  Call Extruder(591.82006)
  MoveL 2707 to (233.6, 37.71, 50.44) mm, rotated rx -180 ry 0 rz 180 deg; joints [-18.033, 13.455, 54.768, 41.267, 27.992, -37.77]
  MoveL 2708 to (233.6, 37.71, 50.44) mm, rotated rx -180 ry 0 rz 180 deg; joints [-18.033, 13.455, 54.768, 41.267, 27.992, -37.77]
  Call Extruder(592.02779)
  MoveL 2709 to (233.9, 37.89, 50.44) mm, rotated rx -180 ry 0 rz 180 deg; joints [-18.041, 13.521, 54.685, 41.26, 28.009, -37.759]
  MoveL 2710 to (233.9, 37.89, 50.44) mm, rotated rx -180 ry 0 rz 180 deg; joints [-18.041, 13.521, 54.685, 41.26, 28.009, -37.759]
  Call Extruder(592.23629)
  MoveL 2711 to (234.21, 38.07, 50.44) mm, rotated rx 180 ry 0 rz 180 deg; joints [-18.049, 13.588, 54.602, 41.254, 28.027, -37.748]
  MoveL 2712 to (234.21, 38.07, 50.44) mm, rotated rx 180 ry 0 rz 180 deg; joints [-18.049, 13.588, 54.602, 41.254, 28.027, -37.748]
  Call Extruder(592.41583)
  MoveL 2713 to (234.45, 38.24, 50.44) mm, rotated rx 180 ry 0 rz 180 deg; joints [-18.06, 13.643, 54.532, 41.254, 28.043, -37.744]
  MoveL 2714 to (234.45, 38.24, 50.44) mm, rotated rx 180 ry 0 rz 180 deg; joints [-18.06, 13.643, 54.532, 41.254, 28.043, -37.744]
  Call Extruder(592.74925)
  MoveL 2715 to (234.9, 38.57, 50.44) mm, rotated rx -180 ry 0 rz -180 deg; joints [-18.079, 13.746, 54.404, 41.255, 28.075, -37.737]
  MoveL 2716 to (234.9, 38.57, 50.44) mm, rotated rx -180 ry 0 rz -180 deg; joints [-18.079, 13.746, 54.404, 41.255, 28.075, -37.737]
  Call Extruder(593.08385)
  MoveL 2717 to (235.35, 38.9, 50.44) mm, rotated rx 180 ry 0 rz -180 deg; joints [-18.099, 13.849, 54.274, 41.255, 28.107, -37.729]
  Call Extruder(593.91180)
  MoveL 2718 to (236.39, 39.81, 50.44) mm, rotated rx -180 ry 0 rz 180 deg; joints [-18.16, 14.097, 53.963, 41.28, 28.192, -37.731]
  Call Extruder(594.73974)
  MoveL 2719 to (237.3, 40.85, 50.44) mm, rotated rx -180 ry 0 rz 180 deg; joints [-18.24, 14.33, 53.668, 41.337, 28.287, -37.762]
  Call Extruder(594.90704)
  MoveL 2720 to (237.47, 41.07, 50.44) mm, rotated rx -180 ry 0 rz 180 deg; joints [-18.258, 14.375, 53.612, 41.353, 28.307, -37.773]
  MoveL 2721 to (237.47, 41.07, 50.44) mm, rotated rx -180 ry 0 rz 180 deg; joints [-18.258, 14.375, 53.612, 41.353, 28.307, -37.773]
  Call Extruder(595.24045)
  MoveL 2722 to (237.79, 41.52, 50.44) mm, rotated rx 180 ry 0 rz 180 deg; joints [-18.295, 14.464, 53.499, 41.385, 28.347, -37.794]
  MoveL 2723 to (237.79, 41.52, 50.44) mm, rotated rx 180 ry 0 rz 180 deg; joints [-18.295, 14.464, 53.499, 41.385, 28.347, -37.794]
  Call Extruder(595.57268)
  MoveL 2724 to (238.12, 41.98, 50.44) mm, rotated rx 180 ry 0 rz 180 deg; joints [-18.332, 14.554, 53.385, 41.417, 28.388, -37.814]
  MoveL 2725 to (238.12, 41.98, 50.44) mm, rotated rx 180 ry 0 rz 180 deg; joints [-18.332, 14.554, 53.385, 41.417, 28.388, -37.814]
  Call Extruder(595.69039)
  MoveL 2726 to (238.22, 42.15, 50.44) mm, rotated rx 180 ry 0 rz 180 deg; joints [-18.346, 14.583, 53.348, 41.432, 28.403, -37.825]
  MoveL 2727 to (238.22, 42.15, 50.44) mm, rotated rx 180 ry 0 rz 180 deg; joints [-18.346, 14.583, 53.348, 41.432, 28.403, -37.825]
  Call Extruder(595.89811)
  MoveL 2728 to (238.4, 42.45, 50.44) mm, rotated rx -180 ry 0 rz 180 deg; joints [-18.373, 14.635, 53.282, 41.458, 28.429, -37.843]
  MoveL 2729 to (238.4, 42.45, 50.44) mm, rotated rx -180 ry 0 rz 180 deg; joints [-18.373, 14.635, 53.282, 41.458, 28.429, -37.843]
  Call Extruder(596.10507)
  MoveL 2730 to (238.57, 42.75, 50.44) mm, rotated rx -180 ry 0 rz -180 deg; joints [-18.399, 14.687, 53.216, 41.485, 28.456, -37.862]
  MoveL 2731 to (238.57, 42.75, 50.44) mm, rotated rx -180 ry 0 rz -180 deg; joints [-18.399, 14.687, 53.216, 41.485, 28.456, -37.862]
  Call Extruder(596.31124)
  MoveL 2732 to (238.75, 43.06, 50.44) mm, rotated rx 180 ry 0 rz 180 deg; joints [-18.425, 14.739, 53.15, 41.511, 28.483, -37.881]
  MoveL 2733 to (238.75, 43.06, 50.44) mm, rotated rx 180 ry 0 rz 180 deg; joints [-18.425, 14.739, 53.15, 41.511, 28.483, -37.881]
  Call Extruder(596.49292)
  MoveL 2734 to (238.89, 43.34, 50.44) mm, rotated rx 180 ry 0 rz 180 deg; joints [-18.45, 14.783, 53.094, 41.537, 28.507, -37.9]
  MoveL 2735 to (238.89, 43.34, 50.44) mm, rotated rx 180 ry 0 rz 180 deg; joints [-18.45, 14.783, 53.094, 41.537, 28.507, -37.9]
  Call Extruder(596.65093)
  MoveL 2736 to (239, 43.58, 50.44) mm, rotated rx -180 ry 0 rz 180 deg; joints [-18.472, 14.819, 53.048, 41.563, 28.528, -37.919]
  MoveL 2737 to (239, 43.58, 50.44) mm, rotated rx -180 ry 0 rz 180 deg; joints [-18.472, 14.819, 53.048, 41.563, 28.528, -37.919]
  Call Extruder(596.80833)
  MoveL 2738 to (239.11, 43.83, 50.44) mm, rotated rx 180 ry 0 rz -180 deg; joints [-18.495, 14.854, 53.003, 41.588, 28.549, -37.939]
  MoveL 2739 to (239.11, 43.83, 50.44) mm, rotated rx 180 ry 0 rz -180 deg; joints [-18.495, 14.854, 53.003, 41.588, 28.549, -37.939]
  Call Extruder(596.98254)
  MoveL 2740 to (239.22, 44.11, 50.44) mm, rotated rx 180 ry 0 rz 180 deg; joints [-18.521, 14.894, 52.953, 41.617, 28.573, -37.961]
  MoveL 2741 to (239.22, 44.11, 50.44) mm, rotated rx 180 ry 0 rz 180 deg; joints [-18.521, 14.894, 52.953, 41.617, 28.573, -37.961]
  Call Extruder(597.15607)
  MoveL 2742 to (239.34, 44.39, 50.44) mm, rotated rx -180 ry 0 rz 180 deg; joints [-18.546, 14.933, 52.902, 41.646, 28.597, -37.983]
  MoveL 2743 to (239.34, 44.39, 50.44) mm, rotated rx -180 ry 0 rz 180 deg; joints [-18.546, 14.933, 52.902, 41.646, 28.597, -37.983]
  Call Extruder(597.26356)
  MoveL 2744 to (239.41, 44.56, 50.44) mm, rotated rx -180 ry 0 rz -180 deg; joints [-18.562, 14.958, 52.871, 41.664, 28.612, -37.996]
  MoveL 2745 to (239.41, 44.56, 50.44) mm, rotated rx -180 ry 0 rz -180 deg; joints [-18.562, 14.958, 52.871, 41.664, 28.612, -37.996]
  Call Extruder(597.37703)
  MoveL 2746 to (239.47, 44.75, 50.44) mm, rotated rx -180 ry 0 rz -180 deg; joints [-18.58, 14.981, 52.841, 41.685, 28.627, -38.013]
  MoveL 2747 to (239.47, 44.75, 50.44) mm, rotated rx -180 ry 0 rz -180 deg; joints [-18.58, 14.981, 52.841, 41.685, 28.627, -38.013]
  Call Extruder(597.49005)
  MoveL 2748 to (239.53, 44.94, 50.44) mm, rotated rx 180 ry 0 rz 180 deg; joints [-18.598, 15.005, 52.811, 41.707, 28.643, -38.03]
  MoveL 2749 to (239.53, 44.94, 50.44) mm, rotated rx 180 ry 0 rz 180 deg; joints [-18.598, 15.005, 52.811, 41.707, 28.643, -38.03]
  Call Extruder(597.60263)
  MoveL 2750 to (239.59, 45.13, 50.44) mm, rotated rx 180 ry 0 rz -180 deg; joints [-18.616, 15.028, 52.781, 41.728, 28.659, -38.046]
  MoveL 2751 to (239.59, 45.13, 50.44) mm, rotated rx 180 ry 0 rz -180 deg; joints [-18.616, 15.028, 52.781, 41.728, 28.659, -38.046]
  Call Extruder(597.71477)
  MoveL 2752 to (239.65, 45.32, 50.44) mm, rotated rx -180 ry 0 rz 180 deg; joints [-18.634, 15.052, 52.751, 41.749, 28.675, -38.063]
  MoveL 2753 to (239.65, 45.32, 50.44) mm, rotated rx -180 ry 0 rz 180 deg; joints [-18.634, 15.052, 52.751, 41.749, 28.675, -38.063]
  Call Extruder(597.82645)
  MoveL 2754 to (239.71, 45.5, 50.44) mm, rotated rx -180 ry 0 rz 180 deg; joints [-18.651, 15.076, 52.721, 41.771, 28.691, -38.079]
  MoveL 2755 to (239.71, 45.5, 50.44) mm, rotated rx -180 ry 0 rz 180 deg; joints [-18.651, 15.076, 52.721, 41.771, 28.691, -38.079]
  Call Extruder(597.95753)
  MoveL 2756 to (239.78, 45.73, 50.44) mm, rotated rx -180 ry 0 rz 180 deg; joints [-18.673, 15.103, 52.686, 41.796, 28.71, -38.099]
  MoveL 2757 to (239.78, 45.73, 50.44) mm, rotated rx -180 ry 0 rz 180 deg; joints [-18.673, 15.103, 52.686, 41.796, 28.71, -38.099]
  Call Extruder(598.08804)
  MoveL 2758 to (239.85, 45.95, 50.44) mm, rotated rx 180 ry 0 rz 180 deg; joints [-18.694, 15.13, 52.651, 41.822, 28.729, -38.12]
  MoveL 2759 to (239.85, 45.95, 50.44) mm, rotated rx 180 ry 0 rz 180 deg; joints [-18.694, 15.13, 52.651, 41.822, 28.729, -38.12]
  Call Extruder(598.21798)
  MoveL 2760 to (239.92, 46.18, 50.44) mm, rotated rx -180 ry 0 rz 180 deg; joints [-18.715, 15.157, 52.616, 41.848, 28.747, -38.14]
  MoveL 2761 to (239.92, 46.18, 50.44) mm, rotated rx -180 ry 0 rz 180 deg; joints [-18.715, 15.157, 52.616, 41.848, 28.747, -38.14]
  Call Extruder(598.34736)
  MoveL 2762 to (239.98, 46.4, 50.44) mm, rotated rx -180 ry 0 rz -180 deg; joints [-18.737, 15.184, 52.581, 41.873, 28.766, -38.159]
  MoveL 2763 to (239.98, 46.4, 50.44) mm, rotated rx -180 ry 0 rz -180 deg; joints [-18.737, 15.184, 52.581, 41.873, 28.766, -38.159]
  Call Extruder(598.46931)
  MoveL 2764 to (240.04, 46.61, 50.44) mm, rotated rx 180 ry 0 rz 180 deg; joints [-18.757, 15.209, 52.55, 41.899, 28.784, -38.18]
  MoveL 2765 to (240.04, 46.61, 50.44) mm, rotated rx 180 ry 0 rz 180 deg; joints [-18.757, 15.209, 52.55, 41.899, 28.784, -38.18]
  Call Extruder(598.58414)
  MoveL 2766 to (240.08, 46.82, 50.44) mm, rotated rx -180 ry 0 rz 180 deg; joints [-18.777, 15.23, 52.522, 41.924, 28.801, -38.2]
  MoveL 2767 to (240.08, 46.82, 50.44) mm, rotated rx -180 ry 0 rz 180 deg; joints [-18.777, 15.23, 52.522, 41.924, 28.801, -38.2]
  Call Extruder(598.69851)
  MoveL 2768 to (240.13, 47.02, 50.44) mm, rotated rx 180 ry 0 rz -180 deg; joints [-18.797, 15.252, 52.495, 41.949, 28.818, -38.22]
  MoveL 2769 to (240.13, 47.02, 50.44) mm, rotated rx 180 ry 0 rz -180 deg; joints [-18.797, 15.252, 52.495, 41.949, 28.818, -38.22]
  Call Extruder(598.81243)
  MoveL 2770 to (240.17, 47.23, 50.44) mm, rotated rx 180 ry 0 rz 180 deg; joints [-18.817, 15.274, 52.467, 41.974, 28.835, -38.24]
  MoveL 2771 to (240.17, 47.23, 50.44) mm, rotated rx 180 ry 0 rz 180 deg; joints [-18.817, 15.274, 52.467, 41.974, 28.835, -38.24]
  Call Extruder(598.92591)
  MoveL 2772 to (240.22, 47.43, 50.44) mm, rotated rx -180 ry 0 rz -180 deg; joints [-18.837, 15.295, 52.439, 42, 28.852, -38.26]
  MoveL 2773 to (240.22, 47.43, 50.44) mm, rotated rx -180 ry 0 rz -180 deg; joints [-18.837, 15.295, 52.439, 42, 28.852, -38.26]
  Call Extruder(599.06319)
  MoveL 2774 to (240.27, 47.68, 50.44) mm, rotated rx -180 ry 0 rz -180 deg; joints [-18.862, 15.321, 52.406, 42.031, 28.873, -38.285]
  MoveL 2775 to (240.27, 47.68, 50.44) mm, rotated rx -180 ry 0 rz -180 deg; joints [-18.862, 15.321, 52.406, 42.031, 28.873, -38.285]
  Call Extruder(599.19986)
  MoveL 2776 to (240.32, 47.93, 50.44) mm, rotated rx 180 ry 0 rz -180 deg; joints [-18.887, 15.347, 52.373, 42.062, 28.893, -38.31]
  MoveL 2777 to (240.32, 47.93, 50.44) mm, rotated rx 180 ry 0 rz -180 deg; joints [-18.887, 15.347, 52.373, 42.062, 28.893, -38.31]
  Call Extruder(599.33592)
  MoveL 2778 to (240.37, 48.18, 50.44) mm, rotated rx 180 ry 0 rz -180 deg; joints [-18.911, 15.372, 52.34, 42.093, 28.914, -38.335]
  MoveL 2779 to (240.37, 48.18, 50.44) mm, rotated rx 180 ry 0 rz -180 deg; joints [-18.911, 15.372, 52.34, 42.093, 28.914, -38.335]
  Call Extruder(599.47137)
  MoveL 2780 to (240.42, 48.43, 50.44) mm, rotated rx 180 ry 0 rz 180 deg; joints [-18.936, 15.398, 52.307, 42.124, 28.934, -38.36]
  MoveL 2781 to (240.42, 48.43, 50.44) mm, rotated rx 180 ry 0 rz 180 deg; joints [-18.936, 15.398, 52.307, 42.124, 28.934, -38.36]
  Call Extruder(599.60622)
  MoveL 2782 to (240.47, 48.68, 50.44) mm, rotated rx -180 ry 0 rz 180 deg; joints [-18.96, 15.424, 52.274, 42.155, 28.955, -38.384]
  MoveL 2783 to (240.47, 48.68, 50.44) mm, rotated rx -180 ry 0 rz 180 deg; joints [-18.96, 15.424, 52.274, 42.155, 28.955, -38.384]
  Call Extruder(599.74045)
  MoveL 2784 to (240.52, 48.92, 50.44) mm, rotated rx -180 ry 0 rz 180 deg; joints [-18.985, 15.45, 52.241, 42.185, 28.976, -38.409]
  MoveL 2785 to (240.52, 48.92, 50.44) mm, rotated rx -180 ry 0 rz 180 deg; joints [-18.985, 15.45, 52.241, 42.185, 28.976, -38.409]
  Call Extruder(599.87407)
  MoveL 2786 to (240.57, 49.17, 50.44) mm, rotated rx -180 ry 0 rz -180 deg; joints [-19.009, 15.475, 52.208, 42.216, 28.996, -38.433]
  MoveL 2787 to (240.57, 49.17, 50.44) mm, rotated rx -180 ry 0 rz -180 deg; joints [-19.009, 15.475, 52.208, 42.216, 28.996, -38.433]
  Call Extruder(600.03618)
  MoveL 2788 to (240.61, 49.48, 50.44) mm, rotated rx -180 ry 0 rz -180 deg; joints [-19.04, 15.505, 52.17, 42.255, 29.022, -38.464]
  MoveL 2789 to (240.61, 49.48, 50.44) mm, rotated rx -180 ry 0 rz -180 deg; joints [-19.04, 15.505, 52.17, 42.255, 29.022, -38.464]
  Call Extruder(600.19756)
  MoveL 2790 to (240.66, 49.79, 50.44) mm, rotated rx -180 ry 0 rz 180 deg; joints [-19.07, 15.534, 52.132, 42.294, 29.047, -38.496]
  MoveL 2791 to (240.66, 49.79, 50.44) mm, rotated rx -180 ry 0 rz 180 deg; joints [-19.07, 15.534, 52.132, 42.294, 29.047, -38.496]
  Call Extruder(600.35821)
  MoveL 2792 to (240.71, 50.09, 50.44) mm, rotated rx 180 ry 0 rz 180 deg; joints [-19.101, 15.564, 52.094, 42.333, 29.072, -38.527]
  MoveL 2793 to (240.71, 50.09, 50.44) mm, rotated rx 180 ry 0 rz 180 deg; joints [-19.101, 15.564, 52.094, 42.333, 29.072, -38.527]
  Call Extruder(600.51814)
  MoveL 2794 to (240.76, 50.4, 50.44) mm, rotated rx 180 ry 0 rz 180 deg; joints [-19.131, 15.593, 52.056, 42.372, 29.097, -38.558]
  MoveL 2795 to (240.76, 50.4, 50.44) mm, rotated rx 180 ry 0 rz 180 deg; joints [-19.131, 15.593, 52.056, 42.372, 29.097, -38.558]
  Call Extruder(600.67734)
  MoveL 2796 to (240.81, 50.7, 50.44) mm, rotated rx -180 ry 0 rz 180 deg; joints [-19.162, 15.623, 52.018, 42.41, 29.123, -38.589]
  MoveL 2797 to (240.81, 50.7, 50.44) mm, rotated rx -180 ry 0 rz 180 deg; joints [-19.162, 15.623, 52.018, 42.41, 29.123, -38.589]
  Call Extruder(600.83580)
  MoveL 2798 to (240.86, 51.01, 50.44) mm, rotated rx 180 ry 0 rz -180 deg; joints [-19.192, 15.652, 51.98, 42.449, 29.148, -38.62]
  MoveL 2799 to (240.86, 51.01, 50.44) mm, rotated rx 180 ry 0 rz -180 deg; joints [-19.192, 15.652, 51.98, 42.449, 29.148, -38.62]
  Call Extruder(601.03468)
  MoveL 2800 to (240.9, 51.4, 50.44) mm, rotated rx 180 ry 0 rz 180 deg; joints [-19.231, 15.687, 51.935, 42.499, 29.18, -38.661]
  MoveL 2801 to (240.9, 51.4, 50.44) mm, rotated rx 180 ry 0 rz 180 deg; joints [-19.231, 15.687, 51.935, 42.499, 29.18, -38.661]
  Call Extruder(601.23269)
  MoveL 2802 to (240.95, 51.78, 50.44) mm, rotated rx 180 ry 0 rz 180 deg; joints [-19.27, 15.722, 51.89, 42.55, 29.212, -38.701]
  MoveL 2803 to (240.95, 51.78, 50.44) mm, rotated rx 180 ry 0 rz 180 deg; joints [-19.27, 15.722, 51.89, 42.55, 29.212, -38.701]
  Call Extruder(601.42983)
  MoveL 2804 to (240.99, 52.17, 50.44) mm, rotated rx 180 ry 0 rz 180 deg; joints [-19.309, 15.757, 51.846, 42.6, 29.244, -38.742]
  MoveL 2805 to (240.99, 52.17, 50.44) mm, rotated rx 180 ry 0 rz 180 deg; joints [-19.309, 15.757, 51.846, 42.6, 29.244, -38.742]
  Call Extruder(601.62610)
  MoveL 2806 to (241.04, 52.56, 50.44) mm, rotated rx -180 ry 0 rz 180 deg; joints [-19.348, 15.791, 51.8, 42.65, 29.276, -38.782]
  MoveL 2807 to (241.04, 52.56, 50.44) mm, rotated rx -180 ry 0 rz 180 deg; joints [-19.348, 15.791, 51.8, 42.65, 29.276, -38.782]
  Call Extruder(601.87181)
  MoveL 2808 to (241.09, 53.05, 50.44) mm, rotated rx 180 ry 0 rz 180 deg; joints [-19.398, 15.833, 51.747, 42.714, 29.316, -38.834]
  MoveL 2809 to (241.09, 53.05, 50.44) mm, rotated rx 180 ry 0 rz 180 deg; joints [-19.398, 15.833, 51.747, 42.714, 29.316, -38.834]
  Call Extruder(602.16658)
  MoveL 2810 to (241.13, 53.64, 50.44) mm, rotated rx 180 ry 0 rz 180 deg; joints [-19.458, 15.882, 51.683, 42.793, 29.364, -38.898]
  MoveL 2811 to (241.13, 53.64, 50.44) mm, rotated rx 180 ry 0 rz 180 deg; joints [-19.458, 15.882, 51.683, 42.793, 29.364, -38.898]
  Call Extruder(602.46002)
  MoveL 2812 to (241.18, 54.23, 50.44) mm, rotated rx 180 ry 0 rz 180 deg; joints [-19.518, 15.931, 51.62, 42.87, 29.412, -38.96]
  MoveL 2813 to (241.18, 54.23, 50.44) mm, rotated rx 180 ry 0 rz 180 deg; joints [-19.518, 15.931, 51.62, 42.87, 29.412, -38.96]
  Call Extruder(602.89337)
  MoveL 2814 to (241.23, 55.1, 50.44) mm, rotated rx 180 ry 0 rz 180 deg; joints [-19.608, 16, 51.531, 42.988, 29.484, -39.056]
  MoveL 2815 to (241.23, 55.1, 50.44) mm, rotated rx 180 ry 0 rz 180 deg; joints [-19.608, 16, 51.531, 42.988, 29.484, -39.056]
  Call Extruder(603.46554)
  MoveL 2816 to (241.27, 56.26, 50.44) mm, rotated rx -180 ry 0 rz 180 deg; joints [-19.728, 16.089, 51.416, 43.145, 29.579, -39.184]
  MoveL 2817 to (241.27, 56.26, 50.44) mm, rotated rx -180 ry 0 rz 180 deg; joints [-19.728, 16.089, 51.416, 43.145, 29.579, -39.184]
  Call Extruder(603.89324)
  MoveL 2818 to (241.29, 57.14, 50.44) mm, rotated rx -180 ry 0 rz 180 deg; joints [-19.819, 16.152, 51.333, 43.264, 29.65, -39.281]
  Call Extruder(645.88687)
  MoveL 2819 to (241.29, 142.86, 50.44) mm, rotated rx 180 ry 0 rz 180 deg; joints [-28.232, 24.205, 40.24, 51.22, 37.359, -44.692]
  MoveL 2820 to (241.29, 142.86, 50.44) mm, rotated rx 180 ry 0 rz 180 deg; joints [-28.232, 24.205, 40.24, 51.22, 37.359, -44.692]
  Call Extruder(646.60231)
  MoveL 2821 to (241.25, 144.32, 50.44) mm, rotated rx 180 ry 0 rz 180 deg; joints [-28.367, 24.38, 39.985, 51.296, 37.504, -44.714]
  MoveL 2822 to (241.25, 144.32, 50.44) mm, rotated rx 180 ry 0 rz 180 deg; joints [-28.367, 24.38, 39.985, 51.296, 37.504, -44.714]
  Call Extruder(647.17705)
  MoveL 2823 to (241.2, 145.48, 50.44) mm, rotated rx -180 ry 0 rz 180 deg; joints [-28.475, 24.517, 39.784, 51.358, 37.62, -44.733]
  MoveL 2824 to (241.2, 145.48, 50.44) mm, rotated rx -180 ry 0 rz 180 deg; joints [-28.475, 24.517, 39.784, 51.358, 37.62, -44.733]
  Call Extruder(647.47049)
  MoveL 2825 to (241.16, 146.07, 50.44) mm, rotated rx -180 ry 0 rz -180 deg; joints [-28.531, 24.582, 39.689, 51.392, 37.679, -44.746]
  MoveL 2826 to (241.16, 146.07, 50.44) mm, rotated rx -180 ry 0 rz -180 deg; joints [-28.531, 24.582, 39.689, 51.392, 37.679, -44.746]
  Call Extruder(647.76527)
  MoveL 2827 to (241.11, 146.66, 50.44) mm, rotated rx -180 ry 0 rz 180 deg; joints [-28.587, 24.647, 39.593, 51.427, 37.737, -44.758]
  MoveL 2828 to (241.11, 146.66, 50.44) mm, rotated rx -180 ry 0 rz 180 deg; joints [-28.587, 24.647, 39.593, 51.427, 37.737, -44.758]
  Call Extruder(648.06138)
  MoveL 2829 to (241.06, 147.25, 50.44) mm, rotated rx 180 ry 0 rz 180 deg; joints [-28.643, 24.713, 39.497, 51.461, 37.796, -44.77]
  MoveL 2830 to (241.06, 147.25, 50.44) mm, rotated rx 180 ry 0 rz 180 deg; joints [-28.643, 24.713, 39.497, 51.461, 37.796, -44.77]
  Call Extruder(648.25765)
  MoveL 2831 to (241.02, 147.64, 50.44) mm, rotated rx 180 ry 0 rz -180 deg; joints [-28.681, 24.752, 39.439, 51.485, 37.834, -44.781]
  MoveL 2832 to (241.02, 147.64, 50.44) mm, rotated rx 180 ry 0 rz -180 deg; joints [-28.681, 24.752, 39.439, 51.485, 37.834, -44.781]
  Call Extruder(648.45479)
  MoveL 2833 to (240.97, 148.02, 50.44) mm, rotated rx 180 ry 0 rz -180 deg; joints [-28.718, 24.792, 39.38, 51.51, 37.872, -44.791]
  MoveL 2834 to (240.97, 148.02, 50.44) mm, rotated rx 180 ry 0 rz -180 deg; joints [-28.718, 24.792, 39.38, 51.51, 37.872, -44.791]
  Call Extruder(648.65280)
  MoveL 2835 to (240.92, 148.41, 50.44) mm, rotated rx -180 ry 0 rz -180 deg; joints [-28.756, 24.832, 39.322, 51.534, 37.91, -44.802]
  MoveL 2836 to (240.92, 148.41, 50.44) mm, rotated rx -180 ry 0 rz -180 deg; joints [-28.756, 24.832, 39.322, 51.534, 37.91, -44.802]
  Call Extruder(648.85167)
  MoveL 2837 to (240.88, 148.8, 50.44) mm, rotated rx 180 ry 0 rz 180 deg; joints [-28.793, 24.872, 39.263, 51.558, 37.948, -44.812]
  MoveL 2838 to (240.88, 148.8, 50.44) mm, rotated rx 180 ry 0 rz 180 deg; joints [-28.793, 24.872, 39.263, 51.558, 37.948, -44.812]
  Call Extruder(649.03075)
  MoveL 2839 to (240.83, 149.14, 50.44) mm, rotated rx -180 ry 0 rz -180 deg; joints [-28.827, 24.906, 39.212, 51.581, 37.982, -44.822]
  MoveL 2840 to (240.83, 149.14, 50.44) mm, rotated rx -180 ry 0 rz -180 deg; joints [-28.827, 24.906, 39.212, 51.581, 37.982, -44.822]
  Call Extruder(649.18995)
  MoveL 2841 to (240.78, 149.45, 50.44) mm, rotated rx -180 ry 0 rz 180 deg; joints [-28.857, 24.935, 39.17, 51.602, 38.011, -44.832]
  MoveL 2842 to (240.78, 149.45, 50.44) mm, rotated rx -180 ry 0 rz 180 deg; joints [-28.857, 24.935, 39.17, 51.602, 38.011, -44.832]
  Call Extruder(649.34987)
  MoveL 2843 to (240.73, 149.76, 50.44) mm, rotated rx 180 ry 0 rz 180 deg; joints [-28.887, 24.964, 39.127, 51.623, 38.041, -44.842]
  MoveL 2844 to (240.73, 149.76, 50.44) mm, rotated rx 180 ry 0 rz 180 deg; joints [-28.887, 24.964, 39.127, 51.623, 38.041, -44.842]
  Call Extruder(649.51052)
  MoveL 2845 to (240.69, 150.06, 50.44) mm, rotated rx 180 ry 0 rz 180 deg; joints [-28.917, 24.993, 39.085, 51.644, 38.071, -44.851]
  MoveL 2846 to (240.69, 150.06, 50.44) mm, rotated rx 180 ry 0 rz 180 deg; joints [-28.917, 24.993, 39.085, 51.644, 38.071, -44.851]
  Call Extruder(649.67190)
  MoveL 2847 to (240.64, 150.37, 50.44) mm, rotated rx 180 ry 0 rz 180 deg; joints [-28.947, 25.022, 39.042, 51.665, 38.101, -44.861]
  MoveL 2848 to (240.64, 150.37, 50.44) mm, rotated rx 180 ry 0 rz 180 deg; joints [-28.947, 25.022, 39.042, 51.665, 38.101, -44.861]
  Call Extruder(649.83401)
  MoveL 2849 to (240.59, 150.67, 50.44) mm, rotated rx 180 ry 0 rz -180 deg; joints [-28.978, 25.051, 38.999, 51.685, 38.13, -44.871]
  MoveL 2850 to (240.59, 150.67, 50.44) mm, rotated rx 180 ry 0 rz -180 deg; joints [-28.978, 25.051, 38.999, 51.685, 38.13, -44.871]
  Call Extruder(649.98221)
  MoveL 2851 to (240.54, 150.95, 50.44) mm, rotated rx 180 ry 0 rz 180 deg; joints [-29.005, 25.076, 38.962, 51.705, 38.157, -44.88]
  MoveL 2852 to (240.54, 150.95, 50.44) mm, rotated rx 180 ry 0 rz 180 deg; joints [-29.005, 25.076, 38.962, 51.705, 38.157, -44.88]
  Call Extruder(650.11644)
  MoveL 2853 to (240.49, 151.2, 50.44) mm, rotated rx -180 ry 0 rz -180 deg; joints [-29.03, 25.098, 38.93, 51.723, 38.181, -44.89]
  MoveL 2854 to (240.49, 151.2, 50.44) mm, rotated rx -180 ry 0 rz -180 deg; joints [-29.03, 25.098, 38.93, 51.723, 38.181, -44.89]
  Call Extruder(650.25129)
  MoveL 2855 to (240.44, 151.45, 50.44) mm, rotated rx 180 ry 0 rz 180 deg; joints [-29.055, 25.119, 38.898, 51.742, 38.205, -44.899]
  MoveL 2856 to (240.44, 151.45, 50.44) mm, rotated rx 180 ry 0 rz 180 deg; joints [-29.055, 25.119, 38.898, 51.742, 38.205, -44.899]
  Call Extruder(650.38674)
  MoveL 2857 to (240.39, 151.7, 50.44) mm, rotated rx 180 ry 0 rz 180 deg; joints [-29.08, 25.141, 38.866, 51.76, 38.229, -44.909]
  MoveL 2858 to (240.39, 151.7, 50.44) mm, rotated rx 180 ry 0 rz 180 deg; joints [-29.08, 25.141, 38.866, 51.76, 38.229, -44.909]
  Call Extruder(650.52280)
  MoveL 2859 to (240.34, 151.95, 50.44) mm, rotated rx 180 ry 0 rz 180 deg; joints [-29.105, 25.162, 38.835, 51.779, 38.253, -44.918]
  MoveL 2860 to (240.34, 151.95, 50.44) mm, rotated rx 180 ry 0 rz 180 deg; joints [-29.105, 25.162, 38.835, 51.779, 38.253, -44.918]
  Call Extruder(650.65947)
  MoveL 2861 to (240.29, 152.2, 50.44) mm, rotated rx -180 ry 0 rz 180 deg; joints [-29.13, 25.184, 38.802, 51.797, 38.277, -44.927]
  MoveL 2862 to (240.29, 152.2, 50.44) mm, rotated rx -180 ry 0 rz 180 deg; joints [-29.13, 25.184, 38.802, 51.797, 38.277, -44.927]
  Call Extruder(650.79675)
  MoveL 2863 to (240.24, 152.45, 50.44) mm, rotated rx 180 ry 0 rz 180 deg; joints [-29.155, 25.205, 38.771, 51.815, 38.301, -44.937]
  MoveL 2864 to (240.24, 152.45, 50.44) mm, rotated rx 180 ry 0 rz 180 deg; joints [-29.155, 25.205, 38.771, 51.815, 38.301, -44.937]
  Call Extruder(650.92242)
  MoveL 2865 to (240.2, 152.67, 50.44) mm, rotated rx 180 ry 0 rz 180 deg; joints [-29.178, 25.225, 38.742, 51.832, 38.323, -44.945]
  MoveL 2866 to (240.2, 152.67, 50.44) mm, rotated rx 180 ry 0 rz 180 deg; joints [-29.178, 25.225, 38.742, 51.832, 38.323, -44.945]
  Call Extruder(651.03634)
  MoveL 2867 to (240.15, 152.88, 50.44) mm, rotated rx 180 ry 0 rz -180 deg; joints [-29.198, 25.241, 38.717, 51.847, 38.343, -44.954]
  MoveL 2868 to (240.15, 152.88, 50.44) mm, rotated rx 180 ry 0 rz -180 deg; joints [-29.198, 25.241, 38.717, 51.847, 38.343, -44.954]
  Call Extruder(651.15072)
  MoveL 2869 to (240.11, 153.08, 50.44) mm, rotated rx 180 ry 0 rz 180 deg; joints [-29.219, 25.258, 38.692, 51.863, 38.362, -44.962]
  MoveL 2870 to (240.11, 153.08, 50.44) mm, rotated rx 180 ry 0 rz 180 deg; joints [-29.219, 25.258, 38.692, 51.863, 38.362, -44.962]
  Call Extruder(651.26555)
  MoveL 2871 to (240.06, 153.28, 50.44) mm, rotated rx 180 ry 0 rz 180 deg; joints [-29.24, 25.275, 38.667, 51.878, 38.382, -44.97]
  MoveL 2872 to (240.06, 153.28, 50.44) mm, rotated rx 180 ry 0 rz 180 deg; joints [-29.24, 25.275, 38.667, 51.878, 38.382, -44.97]
  Call Extruder(651.38083)
  MoveL 2873 to (240.02, 153.49, 50.44) mm, rotated rx 180 ry 0 rz -180 deg; joints [-29.26, 25.292, 38.642, 51.894, 38.401, -44.978]
  MoveL 2874 to (240.02, 153.49, 50.44) mm, rotated rx 180 ry 0 rz -180 deg; joints [-29.26, 25.292, 38.642, 51.894, 38.401, -44.978]
  Call Extruder(651.51021)
  MoveL 2875 to (239.95, 153.71, 50.44) mm, rotated rx 180 ry 0 rz -180 deg; joints [-29.284, 25.306, 38.621, 51.914, 38.422, -44.99]
  MoveL 2876 to (239.95, 153.71, 50.44) mm, rotated rx 180 ry 0 rz -180 deg; joints [-29.284, 25.306, 38.621, 51.914, 38.422, -44.99]
  Call Extruder(651.64015)
  MoveL 2877 to (239.88, 153.94, 50.44) mm, rotated rx 180 ry 0 rz -180 deg; joints [-29.307, 25.32, 38.6, 51.934, 38.443, -45.003]
  MoveL 2878 to (239.88, 153.94, 50.44) mm, rotated rx 180 ry 0 rz -180 deg; joints [-29.307, 25.32, 38.6, 51.934, 38.443, -45.003]
  Call Extruder(651.77066)
  MoveL 2879 to (239.82, 154.16, 50.44) mm, rotated rx -180 ry 0 rz 180 deg; joints [-29.331, 25.335, 38.579, 51.954, 38.464, -45.015]
  MoveL 2880 to (239.82, 154.16, 50.44) mm, rotated rx -180 ry 0 rz 180 deg; joints [-29.331, 25.335, 38.579, 51.954, 38.464, -45.015]
  Call Extruder(651.90174)
  MoveL 2881 to (239.75, 154.38, 50.44) mm, rotated rx 180 ry 0 rz 180 deg; joints [-29.354, 25.349, 38.559, 51.974, 38.485, -45.027]
  MoveL 2882 to (239.75, 154.38, 50.44) mm, rotated rx 180 ry 0 rz 180 deg; joints [-29.354, 25.349, 38.559, 51.974, 38.485, -45.027]
  Call Extruder(652.02338)
  MoveL 2883 to (239.68, 154.59, 50.44) mm, rotated rx -180 ry 0 rz -180 deg; joints [-29.376, 25.361, 38.54, 51.993, 38.504, -45.039]
  MoveL 2884 to (239.68, 154.59, 50.44) mm, rotated rx -180 ry 0 rz -180 deg; joints [-29.376, 25.361, 38.54, 51.993, 38.504, -45.039]
  Call Extruder(652.13550)
  MoveL 2885 to (239.62, 154.78, 50.44) mm, rotated rx 180 ry 0 rz 180 deg; joints [-29.396, 25.372, 38.524, 52.01, 38.521, -45.05]
  MoveL 2886 to (239.62, 154.78, 50.44) mm, rotated rx 180 ry 0 rz 180 deg; joints [-29.396, 25.372, 38.524, 52.01, 38.521, -45.05]
  Call Extruder(652.24807)
  MoveL 2887 to (239.56, 154.97, 50.44) mm, rotated rx -180 ry 0 rz -180 deg; joints [-29.416, 25.383, 38.507, 52.028, 38.539, -45.061]
  MoveL 2888 to (239.56, 154.97, 50.44) mm, rotated rx -180 ry 0 rz -180 deg; joints [-29.416, 25.383, 38.507, 52.028, 38.539, -45.061]
  Call Extruder(652.36108)
  MoveL 2889 to (239.5, 155.15, 50.44) mm, rotated rx 180 ry 0 rz 180 deg; joints [-29.436, 25.394, 38.491, 52.045, 38.556, -45.072]
  MoveL 2890 to (239.5, 155.15, 50.44) mm, rotated rx 180 ry 0 rz 180 deg; joints [-29.436, 25.394, 38.491, 52.045, 38.556, -45.072]
  Call Extruder(652.47454)
  MoveL 2891 to (239.44, 155.34, 50.44) mm, rotated rx -180 ry 0 rz 180 deg; joints [-29.456, 25.405, 38.475, 52.063, 38.574, -45.084]
  MoveL 2892 to (239.44, 155.34, 50.44) mm, rotated rx -180 ry 0 rz 180 deg; joints [-29.456, 25.405, 38.475, 52.063, 38.574, -45.084]
  Call Extruder(652.62218)
  MoveL 2893 to (239.35, 155.58, 50.44) mm, rotated rx 180 ry 0 rz 180 deg; joints [-29.483, 25.416, 38.459, 52.087, 38.596, -45.1]
  MoveL 2894 to (239.35, 155.58, 50.44) mm, rotated rx 180 ry 0 rz 180 deg; joints [-29.483, 25.416, 38.459, 52.087, 38.596, -45.1]
  Call Extruder(652.80452)
  MoveL 2895 to (239.23, 155.87, 50.44) mm, rotated rx -180 ry 0 rz 180 deg; joints [-29.515, 25.427, 38.443, 52.118, 38.622, -45.122]
  MoveL 2896 to (239.23, 155.87, 50.44) mm, rotated rx -180 ry 0 rz 180 deg; joints [-29.515, 25.427, 38.443, 52.118, 38.622, -45.122]
  Call Extruder(652.98761)
  MoveL 2897 to (239.11, 156.17, 50.44) mm, rotated rx 180 ry 0 rz -180 deg; joints [-29.547, 25.438, 38.426, 52.15, 38.648, -45.144]
  MoveL 2898 to (239.11, 156.17, 50.44) mm, rotated rx 180 ry 0 rz -180 deg; joints [-29.547, 25.438, 38.426, 52.15, 38.648, -45.144]
  Call Extruder(653.14533)
  MoveL 2899 to (239, 156.42, 50.44) mm, rotated rx -180 ry 0 rz -180 deg; joints [-29.575, 25.446, 38.414, 52.177, 38.67, -45.163]
  MoveL 2900 to (239, 156.42, 50.44) mm, rotated rx -180 ry 0 rz -180 deg; joints [-29.575, 25.446, 38.414, 52.177, 38.67, -45.163]
  Call Extruder(653.30365)
  MoveL 2901 to (238.89, 156.66, 50.44) mm, rotated rx 180 ry 0 rz 180 deg; joints [-29.603, 25.454, 38.402, 52.204, 38.692, -45.182]
  MoveL 2902 to (238.89, 156.66, 50.44) mm, rotated rx 180 ry 0 rz 180 deg; joints [-29.603, 25.454, 38.402, 52.204, 38.692, -45.182]
  Call Extruder(653.48569)
  MoveL 2903 to (238.75, 156.94, 50.44) mm, rotated rx 180 ry 0 rz 180 deg; joints [-29.635, 25.458, 38.396, 52.239, 38.716, -45.208]
  MoveL 2904 to (238.75, 156.94, 50.44) mm, rotated rx 180 ry 0 rz 180 deg; joints [-29.635, 25.458, 38.396, 52.239, 38.716, -45.208]
  Call Extruder(653.69224)
  MoveL 2905 to (238.57, 157.25, 50.44) mm, rotated rx -180 ry 0 rz -180 deg; joints [-29.671, 25.458, 38.397, 52.279, 38.742, -45.24]
  MoveL 2906 to (238.57, 157.25, 50.44) mm, rotated rx -180 ry 0 rz -180 deg; joints [-29.671, 25.458, 38.397, 52.279, 38.742, -45.24]
  Call Extruder(653.89957)
  MoveL 2907 to (238.4, 157.55, 50.44) mm, rotated rx 180 ry 0 rz 180 deg; joints [-29.707, 25.457, 38.397, 52.32, 38.767, -45.272]
  MoveL 2908 to (238.4, 157.55, 50.44) mm, rotated rx 180 ry 0 rz 180 deg; joints [-29.707, 25.457, 38.397, 52.32, 38.767, -45.272]
  Call Extruder(654.10768)
  MoveL 2909 to (238.22, 157.85, 50.44) mm, rotated rx 180 ry 0 rz 180 deg; joints [-29.743, 25.457, 38.398, 52.361, 38.793, -45.304]
  MoveL 2910 to (238.22, 157.85, 50.44) mm, rotated rx 180 ry 0 rz 180 deg; joints [-29.743, 25.457, 38.398, 52.361, 38.793, -45.304]
  Call Extruder(654.22535)
  MoveL 2911 to (238.12, 158.02, 50.44) mm, rotated rx 180 ry 0 rz -180 deg; joints [-29.764, 25.456, 38.399, 52.384, 38.807, -45.322]
  MoveL 2912 to (238.12, 158.02, 50.44) mm, rotated rx 180 ry 0 rz -180 deg; joints [-29.764, 25.456, 38.399, 52.384, 38.807, -45.322]
  Call Extruder(654.55818)
  MoveL 2913 to (237.79, 158.48, 50.44) mm, rotated rx -180 ry 0 rz 180 deg; joints [-29.821, 25.439, 38.424, 52.457, 38.843, -45.383]
  MoveL 2914 to (237.79, 158.48, 50.44) mm, rotated rx -180 ry 0 rz 180 deg; joints [-29.821, 25.439, 38.424, 52.457, 38.843, -45.383]
  Call Extruder(654.89221)
  MoveL 2915 to (237.47, 158.93, 50.44) mm, rotated rx -180 ry 0 rz 180 deg; joints [-29.878, 25.423, 38.449, 52.529, 38.879, -45.443]
  MoveL 2916 to (237.47, 158.93, 50.44) mm, rotated rx -180 ry 0 rz 180 deg; joints [-29.878, 25.423, 38.449, 52.529, 38.879, -45.443]
  Call Extruder(655.05980)
  MoveL 2917 to (237.3, 159.15, 50.44) mm, rotated rx 180 ry 0 rz 180 deg; joints [-29.907, 25.414, 38.461, 52.565, 38.897, -45.473]
  Call Extruder(655.88912)
  MoveL 2918 to (236.39, 160.19, 50.44) mm, rotated rx -180 ry 0 rz 180 deg; joints [-30.046, 25.338, 38.574, 52.756, 38.974, -45.64]
  Call Extruder(656.52018)
  MoveL 2919 to (235.6, 160.89, 50.44) mm, rotated rx -180 ry 0 rz -180 deg; joints [-30.149, 25.246, 38.71, 52.914, 39.021, -45.785]
  MoveL 2920 to (235.6, 160.89, 50.44) mm, rotated rx -180 ry 0 rz -180 deg; joints [-30.149, 25.246, 38.71, 52.914, 39.021, -45.785]
  Call Extruder(656.71780)
  MoveL 2921 to (235.35, 161.1, 50.44) mm, rotated rx 180 ry 0 rz 180 deg; joints [-30.182, 25.216, 38.755, 52.964, 39.035, -45.831]
  Call Extruder(657.05182)
  MoveL 2922 to (234.9, 161.43, 50.44) mm, rotated rx -180 ry 0 rz 180 deg; joints [-30.234, 25.153, 38.848, 53.052, 39.055, -45.915]
  MoveL 2923 to (234.9, 161.43, 50.44) mm, rotated rx -180 ry 0 rz 180 deg; joints [-30.234, 25.153, 38.848, 53.052, 39.055, -45.915]
  Call Extruder(657.38465)
  MoveL 2924 to (234.45, 161.76, 50.44) mm, rotated rx 180 ry 0 rz 180 deg; joints [-30.287, 25.091, 38.939, 53.139, 39.075, -45.997]
  MoveL 2925 to (234.45, 161.76, 50.44) mm, rotated rx 180 ry 0 rz 180 deg; joints [-30.287, 25.091, 38.939, 53.139, 39.075, -45.997]
  Call Extruder(657.56385)
  MoveL 2926 to (234.21, 161.94, 50.44) mm, rotated rx 180 ry 0 rz -180 deg; joints [-30.316, 25.057, 38.989, 53.187, 39.086, -46.042]
  MoveL 2927 to (234.21, 161.94, 50.44) mm, rotated rx 180 ry 0 rz -180 deg; joints [-30.316, 25.057, 38.989, 53.187, 39.086, -46.042]
  Call Extruder(657.77197)
  MoveL 2928 to (233.9, 162.11, 50.44) mm, rotated rx 180 ry 0 rz 180 deg; joints [-30.347, 25.009, 39.06, 53.244, 39.095, -46.098]
  MoveL 2929 to (233.9, 162.11, 50.44) mm, rotated rx 180 ry 0 rz 180 deg; joints [-30.347, 25.009, 39.06, 53.244, 39.095, -46.098]
  Call Extruder(657.97930)
  MoveL 2930 to (233.6, 162.29, 50.44) mm, rotated rx -180 ry 0 rz 180 deg; joints [-30.379, 24.962, 39.13, 53.301, 39.104, -46.154]
  MoveL 2931 to (233.6, 162.29, 50.44) mm, rotated rx -180 ry 0 rz 180 deg; joints [-30.379, 24.962, 39.13, 53.301, 39.104, -46.154]
  Call Extruder(658.18586)
  MoveL 2932 to (233.29, 162.46, 50.44) mm, rotated rx -180 ry 0 rz 180 deg; joints [-30.41, 24.914, 39.2, 53.358, 39.114, -46.209]
  MoveL 2933 to (233.29, 162.46, 50.44) mm, rotated rx -180 ry 0 rz 180 deg; joints [-30.41, 24.914, 39.2, 53.358, 39.114, -46.209]
  Call Extruder(658.39164)
  MoveL 2934 to (232.99, 162.64, 50.44) mm, rotated rx -180 ry 0 rz 180 deg; joints [-30.442, 24.867, 39.27, 53.414, 39.123, -46.265]
  MoveL 2935 to (232.99, 162.64, 50.44) mm, rotated rx -180 ry 0 rz 180 deg; joints [-30.442, 24.867, 39.27, 53.414, 39.123, -46.265]
  Call Extruder(658.54991)
  MoveL 2936 to (232.74, 162.74, 50.44) mm, rotated rx -180 ry 0 rz 180 deg; joints [-30.464, 24.823, 39.335, 53.459, 39.127, -46.31]
  MoveL 2937 to (232.74, 162.74, 50.44) mm, rotated rx -180 ry 0 rz 180 deg; joints [-30.464, 24.823, 39.335, 53.459, 39.127, -46.31]
  Call Extruder(658.70759)
  MoveL 2938 to (232.49, 162.85, 50.44) mm, rotated rx -180 ry 0 rz 180 deg; joints [-30.487, 24.779, 39.399, 53.505, 39.131, -46.356]
  MoveL 2939 to (232.49, 162.85, 50.44) mm, rotated rx -180 ry 0 rz 180 deg; joints [-30.487, 24.779, 39.399, 53.505, 39.131, -46.356]
  Call Extruder(658.87768)
  MoveL 2940 to (232.22, 162.97, 50.44) mm, rotated rx 180 ry 0 rz 180 deg; joints [-30.511, 24.731, 39.469, 53.553, 39.136, -46.405]
  MoveL 2941 to (232.22, 162.97, 50.44) mm, rotated rx 180 ry 0 rz 180 deg; joints [-30.511, 24.731, 39.469, 53.553, 39.136, -46.405]
  Call Extruder(659.06004)
  MoveL 2942 to (231.93, 163.09, 50.44) mm, rotated rx 180 ry 0 rz 180 deg; joints [-30.538, 24.68, 39.545, 53.606, 39.14, -46.458]
  MoveL 2943 to (231.93, 163.09, 50.44) mm, rotated rx 180 ry 0 rz 180 deg; joints [-30.538, 24.68, 39.545, 53.606, 39.14, -46.458]
  Call Extruder(659.24164)
  MoveL 2944 to (231.64, 163.21, 50.44) mm, rotated rx 180 ry 0 rz 180 deg; joints [-30.564, 24.628, 39.621, 53.658, 39.145, -46.511]
  MoveL 2945 to (231.64, 163.21, 50.44) mm, rotated rx 180 ry 0 rz 180 deg; joints [-30.564, 24.628, 39.621, 53.658, 39.145, -46.511]
  Call Extruder(659.35509)
  MoveL 2946 to (231.45, 163.27, 50.44) mm, rotated rx 180 ry 0 rz 180 deg; joints [-30.579, 24.593, 39.673, 53.691, 39.146, -46.545]
  MoveL 2947 to (231.45, 163.27, 50.44) mm, rotated rx 180 ry 0 rz 180 deg; joints [-30.579, 24.593, 39.673, 53.691, 39.146, -46.545]
  Call Extruder(659.46809)
  MoveL 2948 to (231.26, 163.33, 50.44) mm, rotated rx 180 ry 0 rz 180 deg; joints [-30.595, 24.557, 39.725, 53.724, 39.148, -46.579]
  MoveL 2949 to (231.26, 163.33, 50.44) mm, rotated rx 180 ry 0 rz 180 deg; joints [-30.595, 24.557, 39.725, 53.724, 39.148, -46.579]
  Call Extruder(659.58064)
  MoveL 2950 to (231.07, 163.39, 50.44) mm, rotated rx -180 ry 0 rz 180 deg; joints [-30.61, 24.522, 39.776, 53.757, 39.149, -46.613]
  MoveL 2951 to (231.07, 163.39, 50.44) mm, rotated rx -180 ry 0 rz 180 deg; joints [-30.61, 24.522, 39.776, 53.757, 39.149, -46.613]
  Call Extruder(659.69275)
  MoveL 2952 to (230.88, 163.45, 50.44) mm, rotated rx 180 ry 0 rz 180 deg; joints [-30.625, 24.487, 39.828, 53.791, 39.151, -46.647]
  MoveL 2953 to (230.88, 163.45, 50.44) mm, rotated rx 180 ry 0 rz 180 deg; joints [-30.625, 24.487, 39.828, 53.791, 39.151, -46.647]
  Call Extruder(659.80442)
  MoveL 2954 to (230.69, 163.51, 50.44) mm, rotated rx 180 ry 0 rz 180 deg; joints [-30.641, 24.452, 39.879, 53.823, 39.152, -46.681]
  MoveL 2955 to (230.69, 163.51, 50.44) mm, rotated rx 180 ry 0 rz 180 deg; joints [-30.641, 24.452, 39.879, 53.823, 39.152, -46.681]
  Call Extruder(659.93552)
  MoveL 2956 to (230.47, 163.58, 50.44) mm, rotated rx 180 ry 0 rz 180 deg; joints [-30.659, 24.409, 39.941, 53.862, 39.154, -46.721]
  MoveL 2957 to (230.47, 163.58, 50.44) mm, rotated rx 180 ry 0 rz 180 deg; joints [-30.659, 24.409, 39.941, 53.862, 39.154, -46.721]
  Call Extruder(660.06605)
  MoveL 2958 to (230.25, 163.65, 50.44) mm, rotated rx 180 ry 0 rz 180 deg; joints [-30.677, 24.367, 40.003, 53.901, 39.155, -46.761]
  MoveL 2959 to (230.25, 163.65, 50.44) mm, rotated rx 180 ry 0 rz 180 deg; joints [-30.677, 24.367, 40.003, 53.901, 39.155, -46.761]
  Call Extruder(660.19601)
  MoveL 2960 to (230.02, 163.72, 50.44) mm, rotated rx 180 ry 0 rz 180 deg; joints [-30.694, 24.325, 40.065, 53.94, 39.157, -46.801]
  MoveL 2961 to (230.02, 163.72, 50.44) mm, rotated rx 180 ry 0 rz 180 deg; joints [-30.694, 24.325, 40.065, 53.94, 39.157, -46.801]
  Call Extruder(660.32541)
  MoveL 2962 to (229.8, 163.78, 50.44) mm, rotated rx 180 ry 0 rz 180 deg; joints [-30.712, 24.283, 40.126, 53.979, 39.158, -46.841]
  MoveL 2963 to (229.8, 163.78, 50.44) mm, rotated rx 180 ry 0 rz 180 deg; joints [-30.712, 24.283, 40.126, 53.979, 39.158, -46.841]
  Call Extruder(660.44739)
  MoveL 2964 to (229.59, 163.84, 50.44) mm, rotated rx 180 ry 0 rz 180 deg; joints [-30.729, 24.241, 40.187, 54.015, 39.159, -46.879]
  MoveL 2965 to (229.59, 163.84, 50.44) mm, rotated rx 180 ry 0 rz 180 deg; joints [-30.729, 24.241, 40.187, 54.015, 39.159, -46.879]
  Call Extruder(660.56223)
  MoveL 2966 to (229.38, 163.88, 50.44) mm, rotated rx -180 ry 0 rz 180 deg; joints [-30.744, 24.201, 40.246, 54.05, 39.159, -46.915]
  MoveL 2967 to (229.38, 163.88, 50.44) mm, rotated rx -180 ry 0 rz 180 deg; joints [-30.744, 24.201, 40.246, 54.05, 39.159, -46.915]
  Call Extruder(660.67663)
  MoveL 2968 to (229.18, 163.93, 50.44) mm, rotated rx 180 ry 0 rz -180 deg; joints [-30.758, 24.16, 40.305, 54.084, 39.159, -46.951]
  MoveL 2969 to (229.18, 163.93, 50.44) mm, rotated rx 180 ry 0 rz -180 deg; joints [-30.758, 24.16, 40.305, 54.084, 39.159, -46.951]
  Call Extruder(660.79057)
  MoveL 2970 to (228.97, 163.97, 50.44) mm, rotated rx 180 ry 0 rz 180 deg; joints [-30.773, 24.12, 40.364, 54.119, 39.159, -46.988]
  MoveL 2971 to (228.97, 163.97, 50.44) mm, rotated rx 180 ry 0 rz 180 deg; joints [-30.773, 24.12, 40.364, 54.119, 39.159, -46.988]
  Call Extruder(660.90406)
  MoveL 2972 to (228.77, 164.02, 50.44) mm, rotated rx 180 ry 0 rz 180 deg; joints [-30.788, 24.079, 40.423, 54.153, 39.159, -47.024]
  MoveL 2973 to (228.77, 164.02, 50.44) mm, rotated rx 180 ry 0 rz 180 deg; joints [-30.788, 24.079, 40.423, 54.153, 39.159, -47.024]
  Call Extruder(661.04134)
  MoveL 2974 to (228.52, 164.07, 50.44) mm, rotated rx -180 ry 0 rz 180 deg; joints [-30.806, 24.03, 40.495, 54.195, 39.159, -47.067]
  MoveL 2975 to (228.52, 164.07, 50.44) mm, rotated rx -180 ry 0 rz 180 deg; joints [-30.806, 24.03, 40.495, 54.195, 39.159, -47.067]
  Call Extruder(661.17802)
  MoveL 2976 to (228.27, 164.12, 50.44) mm, rotated rx 180 ry 0 rz 180 deg; joints [-30.823, 23.98, 40.568, 54.236, 39.159, -47.111]
  MoveL 2977 to (228.27, 164.12, 50.44) mm, rotated rx 180 ry 0 rz 180 deg; joints [-30.823, 23.98, 40.568, 54.236, 39.159, -47.111]
  Call Extruder(661.31408)
  MoveL 2978 to (228.02, 164.17, 50.44) mm, rotated rx 180 ry 0 rz 180 deg; joints [-30.841, 23.93, 40.639, 54.278, 39.159, -47.155]
  MoveL 2979 to (228.02, 164.17, 50.44) mm, rotated rx 180 ry 0 rz 180 deg; joints [-30.841, 23.93, 40.639, 54.278, 39.159, -47.155]
  Call Extruder(661.44953)
  MoveL 2980 to (227.77, 164.22, 50.44) mm, rotated rx -180 ry 0 rz -180 deg; joints [-30.859, 23.881, 40.711, 54.319, 39.158, -47.198]
  MoveL 2981 to (227.77, 164.22, 50.44) mm, rotated rx -180 ry 0 rz -180 deg; joints [-30.859, 23.881, 40.711, 54.319, 39.158, -47.198]
  Call Extruder(661.58438)
  MoveL 2982 to (227.52, 164.27, 50.44) mm, rotated rx -180 ry 0 rz 180 deg; joints [-30.877, 23.832, 40.783, 54.36, 39.159, -47.242]
  MoveL 2983 to (227.52, 164.27, 50.44) mm, rotated rx -180 ry 0 rz 180 deg; joints [-30.877, 23.832, 40.783, 54.36, 39.159, -47.242]
  Call Extruder(661.71861)
  MoveL 2984 to (227.27, 164.32, 50.44) mm, rotated rx 180 ry 0 rz 180 deg; joints [-30.895, 23.783, 40.854, 54.402, 39.159, -47.285]
  MoveL 2985 to (227.27, 164.32, 50.44) mm, rotated rx 180 ry 0 rz 180 deg; joints [-30.895, 23.783, 40.854, 54.402, 39.159, -47.285]
  Call Extruder(661.85223)
  MoveL 2986 to (227.02, 164.36, 50.44) mm, rotated rx -180 ry 0 rz 180 deg; joints [-30.912, 23.733, 40.926, 54.443, 39.159, -47.329]
  MoveL 2987 to (227.02, 164.36, 50.44) mm, rotated rx -180 ry 0 rz 180 deg; joints [-30.912, 23.733, 40.926, 54.443, 39.159, -47.329]
  Call Extruder(662.01433)
  MoveL 2988 to (226.72, 164.41, 50.44) mm, rotated rx 180 ry 0 rz 180 deg; joints [-30.933, 23.672, 41.015, 54.493, 39.158, -47.381]
  MoveL 2989 to (226.72, 164.41, 50.44) mm, rotated rx 180 ry 0 rz 180 deg; joints [-30.933, 23.672, 41.015, 54.493, 39.158, -47.381]
  Call Extruder(662.17571)
  MoveL 2990 to (226.41, 164.46, 50.44) mm, rotated rx 180 ry 0 rz 180 deg; joints [-30.954, 23.61, 41.104, 54.542, 39.157, -47.434]
  MoveL 2991 to (226.41, 164.46, 50.44) mm, rotated rx 180 ry 0 rz 180 deg; joints [-30.954, 23.61, 41.104, 54.542, 39.157, -47.434]
  Call Extruder(662.33636)
  MoveL 2992 to (226.11, 164.51, 50.44) mm, rotated rx 180 ry 0 rz 180 deg; joints [-30.975, 23.548, 41.193, 54.592, 39.157, -47.487]
  MoveL 2993 to (226.11, 164.51, 50.44) mm, rotated rx 180 ry 0 rz 180 deg; joints [-30.975, 23.548, 41.193, 54.592, 39.157, -47.487]
  Call Extruder(662.49628)
  MoveL 2994 to (225.8, 164.56, 50.44) mm, rotated rx 180 ry 0 rz 180 deg; joints [-30.995, 23.487, 41.281, 54.641, 39.156, -47.539]
  MoveL 2995 to (225.8, 164.56, 50.44) mm, rotated rx 180 ry 0 rz 180 deg; joints [-30.995, 23.487, 41.281, 54.641, 39.156, -47.539]
  Call Extruder(662.65547)
  MoveL 2996 to (225.5, 164.61, 50.44) mm, rotated rx 180 ry 0 rz 180 deg; joints [-31.016, 23.426, 41.369, 54.691, 39.156, -47.591]
  MoveL 2997 to (225.5, 164.61, 50.44) mm, rotated rx 180 ry 0 rz 180 deg; joints [-31.016, 23.426, 41.369, 54.691, 39.156, -47.591]
  Call Extruder(662.81393)
  MoveL 2998 to (225.19, 164.66, 50.44) mm, rotated rx 180 ry 0 rz 180 deg; joints [-31.037, 23.365, 41.457, 54.74, 39.156, -47.643]
  MoveL 2999 to (225.19, 164.66, 50.44) mm, rotated rx 180 ry 0 rz 180 deg; joints [-31.037, 23.365, 41.457, 54.74, 39.156, -47.643]
  Call Extruder(663.01281)
  MoveL 3000 to (224.8, 164.7, 50.44) mm, rotated rx -180 ry 0 rz 180 deg; joints [-31.062, 23.286, 41.571, 54.801, 39.154, -47.709]
  MoveL 3001 to (224.8, 164.7, 50.44) mm, rotated rx -180 ry 0 rz 180 deg; joints [-31.062, 23.286, 41.571, 54.801, 39.154, -47.709]
  Call Extruder(663.21082)
  MoveL 3002 to (224.42, 164.75, 50.44) mm, rotated rx 180 ry 0 rz 180 deg; joints [-31.087, 23.207, 41.684, 54.863, 39.153, -47.774]
  MoveL 3003 to (224.42, 164.75, 50.44) mm, rotated rx 180 ry 0 rz 180 deg; joints [-31.087, 23.207, 41.684, 54.863, 39.153, -47.774]
  Call Extruder(663.40796)
  MoveL 3004 to (224.03, 164.79, 50.44) mm, rotated rx 180 ry 0 rz 180 deg; joints [-31.112, 23.129, 41.797, 54.924, 39.152, -47.839]
  MoveL 3005 to (224.03, 164.79, 50.44) mm, rotated rx 180 ry 0 rz 180 deg; joints [-31.112, 23.129, 41.797, 54.924, 39.152, -47.839]
  Call Extruder(663.60423)
  MoveL 3006 to (223.64, 164.84, 50.44) mm, rotated rx 180 ry 0 rz -180 deg; joints [-31.137, 23.051, 41.909, 54.985, 39.151, -47.904]
  MoveL 3007 to (223.64, 164.84, 50.44) mm, rotated rx 180 ry 0 rz -180 deg; joints [-31.137, 23.051, 41.909, 54.985, 39.151, -47.904]
  Call Extruder(663.84990)
  MoveL 3008 to (223.15, 164.89, 50.44) mm, rotated rx 180 ry 0 rz 180 deg; joints [-31.168, 22.951, 42.052, 55.061, 39.149, -47.986]
  MoveL 3009 to (223.15, 164.89, 50.44) mm, rotated rx 180 ry 0 rz 180 deg; joints [-31.168, 22.951, 42.052, 55.061, 39.149, -47.986]
  Call Extruder(664.14459)
  MoveL 3010 to (222.56, 164.93, 50.44) mm, rotated rx 180 ry 0 rz 180 deg; joints [-31.204, 22.83, 42.226, 55.152, 39.146, -48.083]
  MoveL 3011 to (222.56, 164.93, 50.44) mm, rotated rx 180 ry 0 rz 180 deg; joints [-31.204, 22.83, 42.226, 55.152, 39.146, -48.083]
  Call Extruder(664.43795)
  MoveL 3012 to (221.97, 164.98, 50.44) mm, rotated rx -180 ry 0 rz -180 deg; joints [-31.24, 22.71, 42.398, 55.242, 39.143, -48.18]
  MoveL 3013 to (221.97, 164.98, 50.44) mm, rotated rx -180 ry 0 rz -180 deg; joints [-31.24, 22.71, 42.398, 55.242, 39.143, -48.18]
  Call Extruder(664.87126)
  MoveL 3014 to (221.1, 165.03, 50.44) mm, rotated rx 180 ry 0 rz 180 deg; joints [-31.292, 22.529, 42.655, 55.375, 39.138, -48.323]
  MoveL 3015 to (221.1, 165.03, 50.44) mm, rotated rx 180 ry 0 rz 180 deg; joints [-31.292, 22.529, 42.655, 55.375, 39.138, -48.323]
  Call Extruder(665.44342)
  MoveL 3016 to (219.94, 165.07, 50.44) mm, rotated rx -180 ry 0 rz 180 deg; joints [-31.36, 22.289, 42.997, 55.548, 39.132, -48.51]
  MoveL 3017 to (219.94, 165.07, 50.44) mm, rotated rx -180 ry 0 rz 180 deg; joints [-31.36, 22.289, 42.997, 55.548, 39.132, -48.51]
  Call Extruder(665.87130)
  MoveL 3018 to (219.06, 165.09, 50.44) mm, rotated rx 180 ry 0 rz 180 deg; joints [-31.409, 22.108, 43.253, 55.677, 39.126, -48.649]
  Call Extruder(782.51995)
  MoveL 3019 to (-19.06, 165.09, 50.44) mm, rotated rx 180 ry 0 rz 180 deg; joints [-51.475, -9.376, 78.454, 74.13, 54.424, -63.957]
  MoveL 3020 to (-19.06, 165.09, 50.44) mm, rotated rx 180 ry 0 rz 180 deg; joints [-51.475, -9.376, 78.454, 74.13, 54.424, -63.957]
  Call Extruder(783.23557)
  MoveL 3021 to (-20.52, 165.05, 50.44) mm, rotated rx 180 ry 0 rz 180 deg; joints [-51.652, -9.51, 78.565, 74.209, 54.589, -63.985]
  MoveL 3022 to (-20.52, 165.05, 50.44) mm, rotated rx 180 ry 0 rz 180 deg; joints [-51.652, -9.51, 78.565, 74.209, 54.589, -63.985]
  Call Extruder(783.81031)
  MoveL 3023 to (-21.68, 165, 50.44) mm, rotated rx 180 ry 0 rz -180 deg; joints [-51.793, -9.618, 78.654, 74.272, 54.721, -64.006]
  MoveL 3024 to (-21.68, 165, 50.44) mm, rotated rx 180 ry 0 rz -180 deg; joints [-51.793, -9.618, 78.654, 74.272, 54.721, -64.006]
  Call Extruder(784.10367)
  MoveL 3025 to (-22.27, 164.96, 50.44) mm, rotated rx 180 ry 0 rz 180 deg; joints [-51.862, -9.676, 78.701, 74.302, 54.785, -64.015]
  MoveL 3026 to (-22.27, 164.96, 50.44) mm, rotated rx 180 ry 0 rz 180 deg; joints [-51.862, -9.676, 78.701, 74.302, 54.785, -64.015]
  Call Extruder(784.39837)
  MoveL 3027 to (-22.86, 164.91, 50.44) mm, rotated rx 180 ry 0 rz -180 deg; joints [-51.931, -9.733, 78.748, 74.332, 54.85, -64.025]
  MoveL 3028 to (-22.86, 164.91, 50.44) mm, rotated rx 180 ry 0 rz -180 deg; joints [-51.931, -9.733, 78.748, 74.332, 54.85, -64.025]
  Call Extruder(784.69439)
  MoveL 3029 to (-23.45, 164.86, 50.44) mm, rotated rx 180 ry 0 rz -180 deg; joints [-52.001, -9.79, 78.795, 74.362, 54.916, -64.034]
  MoveL 3030 to (-23.45, 164.86, 50.44) mm, rotated rx 180 ry 0 rz -180 deg; joints [-52.001, -9.79, 78.795, 74.362, 54.916, -64.034]
  Call Extruder(784.89067)
  MoveL 3031 to (-23.83, 164.82, 50.44) mm, rotated rx 180 ry 0 rz 180 deg; joints [-52.045, -9.829, 78.827, 74.381, 54.958, -64.039]
  MoveL 3032 to (-23.83, 164.82, 50.44) mm, rotated rx 180 ry 0 rz 180 deg; joints [-52.045, -9.829, 78.827, 74.381, 54.958, -64.039]
  Call Extruder(785.08781)
  MoveL 3033 to (-24.22, 164.77, 50.44) mm, rotated rx 180 ry 0 rz 180 deg; joints [-52.089, -9.868, 78.859, 74.4, 54.999, -64.045]
  MoveL 3034 to (-24.22, 164.77, 50.44) mm, rotated rx 180 ry 0 rz 180 deg; joints [-52.089, -9.868, 78.859, 74.4, 54.999, -64.045]
  Call Extruder(785.28582)
  MoveL 3035 to (-24.61, 164.73, 50.44) mm, rotated rx 180 ry 0 rz 180 deg; joints [-52.134, -9.908, 78.891, 74.419, 55.041, -64.05]
  MoveL 3036 to (-24.61, 164.73, 50.44) mm, rotated rx 180 ry 0 rz 180 deg; joints [-52.134, -9.908, 78.891, 74.419, 55.041, -64.05]
  Call Extruder(785.48469)
  MoveL 3037 to (-25, 164.68, 50.44) mm, rotated rx 180 ry 0 rz 180 deg; joints [-52.178, -9.947, 78.923, 74.438, 55.083, -64.055]
  MoveL 3038 to (-25, 164.68, 50.44) mm, rotated rx 180 ry 0 rz 180 deg; joints [-52.178, -9.947, 78.923, 74.438, 55.083, -64.055]
  Call Extruder(785.66377)
  MoveL 3039 to (-25.34, 164.63, 50.44) mm, rotated rx 180 ry 0 rz 180 deg; joints [-52.218, -9.982, 78.953, 74.455, 55.12, -64.06]
  MoveL 3040 to (-25.34, 164.63, 50.44) mm, rotated rx 180 ry 0 rz 180 deg; joints [-52.218, -9.982, 78.953, 74.455, 55.12, -64.06]
  Call Extruder(785.82297)
  MoveL 3041 to (-25.65, 164.58, 50.44) mm, rotated rx 180 ry 0 rz -180 deg; joints [-52.251, -10.015, 78.979, 74.469, 55.152, -64.063]
  MoveL 3042 to (-25.65, 164.58, 50.44) mm, rotated rx 180 ry 0 rz -180 deg; joints [-52.251, -10.015, 78.979, 74.469, 55.152, -64.063]
  Call Extruder(785.98289)
  MoveL 3043 to (-25.96, 164.53, 50.44) mm, rotated rx -180 ry 0 rz 180 deg; joints [-52.286, -10.047, 79.005, 74.483, 55.184, -64.066]
  MoveL 3044 to (-25.96, 164.53, 50.44) mm, rotated rx -180 ry 0 rz 180 deg; joints [-52.286, -10.047, 79.005, 74.483, 55.184, -64.066]
  Call Extruder(786.14354)
  MoveL 3045 to (-26.26, 164.49, 50.44) mm, rotated rx -180 ry 0 rz 180 deg; joints [-52.32, -10.079, 79.031, 74.497, 55.217, -64.07]
  MoveL 3046 to (-26.26, 164.49, 50.44) mm, rotated rx -180 ry 0 rz 180 deg; joints [-52.32, -10.079, 79.031, 74.497, 55.217, -64.07]
  Call Extruder(786.30492)
  MoveL 3047 to (-26.57, 164.44, 50.44) mm, rotated rx 180 ry 0 rz 180 deg; joints [-52.354, -10.111, 79.057, 74.511, 55.249, -64.073]
  MoveL 3048 to (-26.57, 164.44, 50.44) mm, rotated rx 180 ry 0 rz 180 deg; joints [-52.354, -10.111, 79.057, 74.511, 55.249, -64.073]
  Call Extruder(786.46703)
  MoveL 3049 to (-26.87, 164.39, 50.44) mm, rotated rx 180 ry 0 rz 180 deg; joints [-52.388, -10.143, 79.084, 74.525, 55.281, -64.077]
  MoveL 3050 to (-26.87, 164.39, 50.44) mm, rotated rx 180 ry 0 rz 180 deg; joints [-52.388, -10.143, 79.084, 74.525, 55.281, -64.077]
  Call Extruder(786.61523)
  MoveL 3051 to (-27.15, 164.34, 50.44) mm, rotated rx -180 ry 0 rz 180 deg; joints [-52.418, -10.173, 79.108, 74.538, 55.31, -64.079]
  MoveL 3052 to (-27.15, 164.34, 50.44) mm, rotated rx -180 ry 0 rz 180 deg; joints [-52.418, -10.173, 79.108, 74.538, 55.31, -64.079]
  Call Extruder(786.74946)
  MoveL 3053 to (-27.4, 164.29, 50.44) mm, rotated rx -180 ry 0 rz 180 deg; joints [-52.445, -10.2, 79.13, 74.549, 55.336, -64.082]
  MoveL 3054 to (-27.4, 164.29, 50.44) mm, rotated rx -180 ry 0 rz 180 deg; joints [-52.445, -10.2, 79.13, 74.549, 55.336, -64.082]
  Call Extruder(786.88430)
  MoveL 3055 to (-27.65, 164.24, 50.44) mm, rotated rx 180 ry 0 rz -180 deg; joints [-52.472, -10.227, 79.152, 74.56, 55.361, -64.084]
  MoveL 3056 to (-27.65, 164.24, 50.44) mm, rotated rx 180 ry 0 rz -180 deg; joints [-52.472, -10.227, 79.152, 74.56, 55.361, -64.084]
  Call Extruder(787.01975)
  MoveL 3057 to (-27.9, 164.19, 50.44) mm, rotated rx 180 ry 0 rz 180 deg; joints [-52.499, -10.254, 79.174, 74.571, 55.387, -64.086]
  MoveL 3058 to (-27.9, 164.19, 50.44) mm, rotated rx 180 ry 0 rz 180 deg; joints [-52.499, -10.254, 79.174, 74.571, 55.387, -64.086]
  Call Extruder(787.15582)
  MoveL 3059 to (-28.15, 164.14, 50.44) mm, rotated rx 180 ry 0 rz 180 deg; joints [-52.526, -10.281, 79.196, 74.582, 55.413, -64.088]
  MoveL 3060 to (-28.15, 164.14, 50.44) mm, rotated rx 180 ry 0 rz 180 deg; joints [-52.526, -10.281, 79.196, 74.582, 55.413, -64.088]
  Call Extruder(787.29249)
  MoveL 3061 to (-28.4, 164.09, 50.44) mm, rotated rx 180 ry 0 rz -180 deg; joints [-52.553, -10.309, 79.218, 74.593, 55.438, -64.09]
  MoveL 3062 to (-28.4, 164.09, 50.44) mm, rotated rx 180 ry 0 rz -180 deg; joints [-52.553, -10.309, 79.218, 74.593, 55.438, -64.09]
  Call Extruder(787.42977)
  MoveL 3063 to (-28.64, 164.04, 50.44) mm, rotated rx 180 ry 0 rz 180 deg; joints [-52.58, -10.336, 79.24, 74.604, 55.464, -64.092]
  MoveL 3064 to (-28.64, 164.04, 50.44) mm, rotated rx 180 ry 0 rz 180 deg; joints [-52.58, -10.336, 79.24, 74.604, 55.464, -64.092]
  Call Extruder(787.55544)
  MoveL 3065 to (-28.87, 164, 50.44) mm, rotated rx -180 ry 0 rz 180 deg; joints [-52.605, -10.361, 79.26, 74.613, 55.487, -64.094]
  MoveL 3066 to (-28.87, 164, 50.44) mm, rotated rx -180 ry 0 rz 180 deg; joints [-52.605, -10.361, 79.26, 74.613, 55.487, -64.094]
  Call Extruder(787.66938)
  MoveL 3067 to (-29.08, 163.95, 50.44) mm, rotated rx -180 ry 0 rz 180 deg; joints [-52.627, -10.383, 79.279, 74.622, 55.508, -64.096]
  MoveL 3068 to (-29.08, 163.95, 50.44) mm, rotated rx -180 ry 0 rz 180 deg; joints [-52.627, -10.383, 79.279, 74.622, 55.508, -64.096]
  Call Extruder(787.78378)
  MoveL 3069 to (-29.28, 163.91, 50.44) mm, rotated rx -180 ry 0 rz 180 deg; joints [-52.649, -10.406, 79.297, 74.631, 55.529, -64.097]
  MoveL 3070 to (-29.28, 163.91, 50.44) mm, rotated rx -180 ry 0 rz 180 deg; joints [-52.649, -10.406, 79.297, 74.631, 55.529, -64.097]
  Call Extruder(787.89862)
  MoveL 3071 to (-29.48, 163.86, 50.44) mm, rotated rx 180 ry 0 rz 180 deg; joints [-52.67, -10.429, 79.315, 74.64, 55.55, -64.099]
  MoveL 3072 to (-29.48, 163.86, 50.44) mm, rotated rx 180 ry 0 rz 180 deg; joints [-52.67, -10.429, 79.315, 74.64, 55.55, -64.099]
  Call Extruder(788.01392)
  MoveL 3073 to (-29.69, 163.82, 50.44) mm, rotated rx 180 ry 0 rz 180 deg; joints [-52.692, -10.451, 79.334, 74.648, 55.57, -64.1]
  MoveL 3074 to (-29.69, 163.82, 50.44) mm, rotated rx 180 ry 0 rz 180 deg; joints [-52.692, -10.451, 79.334, 74.648, 55.57, -64.1]
  Call Extruder(788.14332)
  MoveL 3075 to (-29.91, 163.75, 50.44) mm, rotated rx 180 ry 0 rz 180 deg; joints [-52.714, -10.478, 79.356, 74.657, 55.592, -64.101]
  MoveL 3076 to (-29.91, 163.75, 50.44) mm, rotated rx 180 ry 0 rz 180 deg; joints [-52.714, -10.478, 79.356, 74.657, 55.592, -64.101]
  Call Extruder(788.27328)
  MoveL 3077 to (-30.14, 163.68, 50.44) mm, rotated rx 180 ry 0 rz -180 deg; joints [-52.737, -10.505, 79.377, 74.665, 55.613, -64.101]
  MoveL 3078 to (-30.14, 163.68, 50.44) mm, rotated rx 180 ry 0 rz -180 deg; joints [-52.737, -10.505, 79.377, 74.665, 55.613, -64.101]
  Call Extruder(788.40380)
  MoveL 3079 to (-30.36, 163.62, 50.44) mm, rotated rx -180 ry 0 rz 180 deg; joints [-52.759, -10.532, 79.399, 74.673, 55.634, -64.102]
  MoveL 3080 to (-30.36, 163.62, 50.44) mm, rotated rx -180 ry 0 rz 180 deg; joints [-52.759, -10.532, 79.399, 74.673, 55.634, -64.102]
  Call Extruder(788.53489)
  MoveL 3081 to (-30.58, 163.55, 50.44) mm, rotated rx 180 ry 0 rz 180 deg; joints [-52.781, -10.559, 79.421, 74.682, 55.656, -64.102]
  MoveL 3082 to (-30.58, 163.55, 50.44) mm, rotated rx 180 ry 0 rz 180 deg; joints [-52.781, -10.559, 79.421, 74.682, 55.656, -64.102]
  Call Extruder(788.65654)
  MoveL 3083 to (-30.79, 163.48, 50.44) mm, rotated rx -180 ry 0 rz -180 deg; joints [-52.801, -10.584, 79.441, 74.689, 55.675, -64.103]
  MoveL 3084 to (-30.79, 163.48, 50.44) mm, rotated rx -180 ry 0 rz -180 deg; joints [-52.801, -10.584, 79.441, 74.689, 55.675, -64.103]
  Call Extruder(788.76865)
  MoveL 3085 to (-30.98, 163.42, 50.44) mm, rotated rx -180 ry 0 rz 180 deg; joints [-52.82, -10.607, 79.459, 74.696, 55.693, -64.103]
  MoveL 3086 to (-30.98, 163.42, 50.44) mm, rotated rx -180 ry 0 rz 180 deg; joints [-52.82, -10.607, 79.459, 74.696, 55.693, -64.103]
  Call Extruder(788.88121)
  MoveL 3087 to (-31.17, 163.36, 50.44) mm, rotated rx -180 ry 0 rz 180 deg; joints [-52.838, -10.63, 79.478, 74.703, 55.711, -64.103]
  MoveL 3088 to (-31.17, 163.36, 50.44) mm, rotated rx -180 ry 0 rz 180 deg; joints [-52.838, -10.63, 79.478, 74.703, 55.711, -64.103]
  Call Extruder(788.99421)
  MoveL 3089 to (-31.35, 163.3, 50.44) mm, rotated rx 180 ry 0 rz 180 deg; joints [-52.856, -10.653, 79.496, 74.709, 55.728, -64.103]
  MoveL 3090 to (-31.35, 163.3, 50.44) mm, rotated rx 180 ry 0 rz 180 deg; joints [-52.856, -10.653, 79.496, 74.709, 55.728, -64.103]
  Call Extruder(789.10766)
  MoveL 3091 to (-31.54, 163.24, 50.44) mm, rotated rx -180 ry 0 rz -180 deg; joints [-52.875, -10.676, 79.515, 74.716, 55.746, -64.104]
  MoveL 3092 to (-31.54, 163.24, 50.44) mm, rotated rx -180 ry 0 rz -180 deg; joints [-52.875, -10.676, 79.515, 74.716, 55.746, -64.104]
  Call Extruder(789.25531)
  MoveL 3093 to (-31.78, 163.15, 50.44) mm, rotated rx 180 ry 0 rz 180 deg; joints [-52.897, -10.707, 79.54, 74.724, 55.768, -64.103]
  MoveL 3094 to (-31.78, 163.15, 50.44) mm, rotated rx 180 ry 0 rz 180 deg; joints [-52.897, -10.707, 79.54, 74.724, 55.768, -64.103]
  Call Extruder(789.43766)
  MoveL 3095 to (-32.07, 163.03, 50.44) mm, rotated rx 180 ry 0 rz 180 deg; joints [-52.923, -10.746, 79.571, 74.733, 55.793, -64.102]
  MoveL 3096 to (-32.07, 163.03, 50.44) mm, rotated rx 180 ry 0 rz 180 deg; joints [-52.923, -10.746, 79.571, 74.733, 55.793, -64.102]
  Call Extruder(789.62078)
  MoveL 3097 to (-32.37, 162.91, 50.44) mm, rotated rx 180 ry 0 rz 180 deg; joints [-52.949, -10.784, 79.602, 74.741, 55.819, -64.101]
  MoveL 3098 to (-32.37, 162.91, 50.44) mm, rotated rx 180 ry 0 rz 180 deg; joints [-52.949, -10.784, 79.602, 74.741, 55.819, -64.101]
  Call Extruder(789.77845)
  MoveL 3099 to (-32.62, 162.8, 50.44) mm, rotated rx 180 ry 0 rz 180 deg; joints [-52.971, -10.818, 79.629, 74.749, 55.84, -64.1]
  MoveL 3100 to (-32.62, 162.8, 50.44) mm, rotated rx 180 ry 0 rz 180 deg; joints [-52.971, -10.818, 79.629, 74.749, 55.84, -64.1]
  Call Extruder(789.93673)
  MoveL 3101 to (-32.87, 162.69, 50.44) mm, rotated rx -180 ry 0 rz 180 deg; joints [-52.993, -10.851, 79.655, 74.756, 55.862, -64.098]
  MoveL 3102 to (-32.87, 162.69, 50.44) mm, rotated rx -180 ry 0 rz 180 deg; joints [-52.993, -10.851, 79.655, 74.756, 55.862, -64.098]
  Call Extruder(790.11874)
  MoveL 3103 to (-33.14, 162.55, 50.44) mm, rotated rx -180 ry 0 rz 180 deg; joints [-53.015, -10.891, 79.687, 74.762, 55.884, -64.096]
  MoveL 3104 to (-33.14, 162.55, 50.44) mm, rotated rx -180 ry 0 rz 180 deg; joints [-53.015, -10.891, 79.687, 74.762, 55.884, -64.096]
  Call Extruder(790.32530)
  MoveL 3105 to (-33.45, 162.37, 50.44) mm, rotated rx 180 ry 0 rz 180 deg; joints [-53.038, -10.937, 79.724, 74.768, 55.906, -64.092]
  MoveL 3106 to (-33.45, 162.37, 50.44) mm, rotated rx 180 ry 0 rz 180 deg; joints [-53.038, -10.937, 79.724, 74.768, 55.906, -64.092]
  Call Extruder(790.53263)
  MoveL 3107 to (-33.75, 162.2, 50.44) mm, rotated rx 180 ry 0 rz 180 deg; joints [-53.06, -10.982, 79.76, 74.774, 55.929, -64.088]
  MoveL 3108 to (-33.75, 162.2, 50.44) mm, rotated rx 180 ry 0 rz 180 deg; joints [-53.06, -10.982, 79.76, 74.774, 55.929, -64.088]
  Call Extruder(790.74074)
  MoveL 3109 to (-34.05, 162.02, 50.44) mm, rotated rx 180 ry 0 rz 180 deg; joints [-53.083, -11.028, 79.797, 74.78, 55.951, -64.084]
  MoveL 3110 to (-34.05, 162.02, 50.44) mm, rotated rx 180 ry 0 rz 180 deg; joints [-53.083, -11.028, 79.797, 74.78, 55.951, -64.084]
  Call Extruder(790.85846)
  MoveL 3111 to (-34.23, 161.92, 50.44) mm, rotated rx -180 ry 0 rz 180 deg; joints [-53.095, -11.054, 79.817, 74.783, 55.964, -64.081]
  MoveL 3112 to (-34.23, 161.92, 50.44) mm, rotated rx -180 ry 0 rz 180 deg; joints [-53.095, -11.054, 79.817, 74.783, 55.964, -64.081]
  Call Extruder(791.19129)
  MoveL 3113 to (-34.68, 161.6, 50.44) mm, rotated rx 180 ry 0 rz 180 deg; joints [-53.122, -11.129, 79.877, 74.787, 55.992, -64.071]
  MoveL 3114 to (-34.68, 161.6, 50.44) mm, rotated rx 180 ry 0 rz 180 deg; joints [-53.122, -11.129, 79.877, 74.787, 55.992, -64.071]
  Call Extruder(791.52530)
  MoveL 3115 to (-35.13, 161.27, 50.44) mm, rotated rx 180 ry 0 rz 180 deg; joints [-53.149, -11.205, 79.937, 74.792, 56.021, -64.061]
  MoveL 3116 to (-35.13, 161.27, 50.44) mm, rotated rx 180 ry 0 rz 180 deg; joints [-53.149, -11.205, 79.937, 74.792, 56.021, -64.061]
  Call Extruder(791.69289)
  MoveL 3117 to (-35.35, 161.1, 50.44) mm, rotated rx 180 ry 0 rz -180 deg; joints [-53.163, -11.242, 79.967, 74.794, 56.035, -64.056]
  Call Extruder(792.52220)
  MoveL 3118 to (-36.39, 160.19, 50.44) mm, rotated rx 180 ry 0 rz 180 deg; joints [-53.209, -11.433, 80.118, 74.793, 56.087, -64.024]
  Call Extruder(793.04443)
  MoveL 3119 to (-36.97, 159.54, 50.44) mm, rotated rx 180 ry 0 rz 180 deg; joints [-53.221, -11.555, 80.215, 74.782, 56.105, -63.997]
  Set speed (130.0 mm/s)
  MoveL 3120 to (-38.97, 156.79, 50.44) mm, rotated rx 180 ry 0 rz 180 deg; joints [-53.214, -12.034, 80.59, 74.711, 56.126, -63.874]
  MoveL 3121 to (-38.97, 156.78, 59.84) mm, rotated rx 180 ry 0 rz 180 deg; joints [-53.214, -12.901, 82.814, 75.597, 55.778, -65.457]
  Call Extruder(791.04443)
  Set speed (40.0 mm/s)
  MoveL 3122 to (-38.97, 156.78, 59.84) mm, rotated rx 180 ry 0 rz 180 deg; joints [-53.214, -12.901, 82.814, 75.597, 55.778, -65.457]
  Call Extruder(0.00000)
  Set speed (130.0 mm/s)
  MoveL 3123 to (-31.64, 163.21, 59.84) mm, rotated rx -180 ry 0 rz 180 deg; joints [-52.884, -11.554, 81.764, 75.629, 55.404, -65.713]
  Call Extruder(2.00000)
  Set speed (40.0 mm/s)
  MoveL 3124 to (-31.64, 163.21, 59.84) mm, rotated rx -180 ry 0 rz 180 deg; joints [-52.884, -11.554, 81.764, 75.629, 55.404, -65.713]
  Set speed (30.0 mm/s)
  MoveL 3125 to (-31.64, 163.21, 59.84) mm, rotated rx -180 ry 0 rz 180 deg; joints [-52.884, -11.554, 81.764, 75.629, 55.404, -65.713]
  Call Extruder(2.18198)
  MoveL 3126 to (-31.93, 163.09, 59.84) mm, rotated rx 180 ry 0 rz 180 deg; joints [-52.91, -11.593, 81.795, 75.637, 55.429, -65.711]
  MoveL 3127 to (-31.93, 163.09, 59.84) mm, rotated rx 180 ry 0 rz 180 deg; joints [-52.91, -11.593, 81.795, 75.637, 55.429, -65.711]
  Call Extruder(2.36471)
  MoveL 3128 to (-32.22, 162.96, 59.84) mm, rotated rx -180 ry 0 rz 180 deg; joints [-52.936, -11.632, 81.825, 75.645, 55.455, -65.709]
  MoveL 3129 to (-32.22, 162.96, 59.84) mm, rotated rx -180 ry 0 rz 180 deg; joints [-52.936, -11.632, 81.825, 75.645, 55.455, -65.709]
  Call Extruder(2.53513)
  MoveL 3130 to (-32.49, 162.85, 59.84) mm, rotated rx 180 ry 0 rz 180 deg; joints [-52.96, -11.668, 81.854, 75.651, 55.479, -65.707]
  MoveL 3131 to (-32.49, 162.85, 59.84) mm, rotated rx 180 ry 0 rz 180 deg; joints [-52.96, -11.668, 81.854, 75.651, 55.479, -65.707]
  Call Extruder(2.69310)
  MoveL 3132 to (-32.74, 162.74, 59.84) mm, rotated rx 180 ry 0 rz -180 deg; joints [-52.982, -11.701, 81.88, 75.658, 55.501, -65.705]
  MoveL 3133 to (-32.74, 162.74, 59.84) mm, rotated rx 180 ry 0 rz -180 deg; joints [-52.982, -11.701, 81.88, 75.658, 55.501, -65.705]
  Call Extruder(2.85168)
  MoveL 3134 to (-32.99, 162.64, 59.84) mm, rotated rx 180 ry 0 rz 180 deg; joints [-53.004, -11.734, 81.906, 75.664, 55.522, -65.703]
  MoveL 3135 to (-32.99, 162.64, 59.84) mm, rotated rx 180 ry 0 rz 180 deg; joints [-53.004, -11.734, 81.906, 75.664, 55.522, -65.703]
  Call Extruder(3.05785)
  MoveL 3136 to (-33.29, 162.46, 59.84) mm, rotated rx -180 ry 0 rz 180 deg; joints [-53.026, -11.78, 81.942, 75.669, 55.545, -65.697]
  MoveL 3137 to (-33.29, 162.46, 59.84) mm, rotated rx -180 ry 0 rz 180 deg; joints [-53.026, -11.78, 81.942, 75.669, 55.545, -65.697]
  Call Extruder(3.26479)
  MoveL 3138 to (-33.6, 162.29, 59.84) mm, rotated rx 180 ry 0 rz 180 deg; joints [-53.049, -11.826, 81.979, 75.673, 55.568, -65.692]
  MoveL 3139 to (-33.6, 162.29, 59.84) mm, rotated rx 180 ry 0 rz 180 deg; joints [-53.049, -11.826, 81.979, 75.673, 55.568, -65.692]
  Call Extruder(3.47251)
  MoveL 3140 to (-33.9, 162.11, 59.84) mm, rotated rx 180 ry 0 rz 180 deg; joints [-53.071, -11.872, 82.014, 75.678, 55.591, -65.687]
  MoveL 3141 to (-33.9, 162.11, 59.84) mm, rotated rx 180 ry 0 rz 180 deg; joints [-53.071, -11.872, 82.014, 75.678, 55.591, -65.687]
  Call Extruder(3.68101)
  MoveL 3142 to (-34.21, 161.94, 59.84) mm, rotated rx 180 ry 0 rz 180 deg; joints [-53.094, -11.917, 82.05, 75.683, 55.614, -65.682]
  MoveL 3143 to (-34.21, 161.94, 59.84) mm, rotated rx 180 ry 0 rz 180 deg; joints [-53.094, -11.917, 82.05, 75.683, 55.614, -65.682]
  Call Extruder(3.86055)
  MoveL 3144 to (-34.45, 161.76, 59.84) mm, rotated rx 180 ry 0 rz 180 deg; joints [-53.109, -11.958, 82.082, 75.684, 55.63, -65.676]
  MoveL 3145 to (-34.45, 161.76, 59.84) mm, rotated rx 180 ry 0 rz 180 deg; joints [-53.109, -11.958, 82.082, 75.684, 55.63, -65.676]
  Call Extruder(4.19399)
  MoveL 3146 to (-34.9, 161.43, 59.84) mm, rotated rx -180 ry 0 rz 180 deg; joints [-53.135, -12.033, 82.141, 75.687, 55.658, -65.664]
  MoveL 3147 to (-34.9, 161.43, 59.84) mm, rotated rx -180 ry 0 rz 180 deg; joints [-53.135, -12.033, 82.141, 75.687, 55.658, -65.664]
  Call Extruder(4.52861)
  MoveL 3148 to (-35.35, 161.1, 59.84) mm, rotated rx 180 ry 0 rz -180 deg; joints [-53.163, -12.109, 82.2, 75.69, 55.687, -65.653]
  Call Extruder(5.35652)
  MoveL 3149 to (-36.39, 160.19, 59.84) mm, rotated rx 180 ry 0 rz 180 deg; joints [-53.209, -12.3, 82.349, 75.685, 55.74, -65.616]
  Call Extruder(6.18445)
  MoveL 3150 to (-37.3, 159.15, 59.84) mm, rotated rx 180 ry 0 rz 180 deg; joints [-53.227, -12.494, 82.5, 75.666, 55.767, -65.571]
  Call Extruder(6.35176)
  MoveL 3151 to (-37.47, 158.93, 59.84) mm, rotated rx 180 ry 0 rz -180 deg; joints [-53.227, -12.533, 82.53, 75.659, 55.769, -65.56]
  MoveL 3152 to (-37.47, 158.93, 59.84) mm, rotated rx 180 ry 0 rz -180 deg; joints [-53.227, -12.533, 82.53, 75.659, 55.769, -65.56]
  Call Extruder(6.68519)
  MoveL 3153 to (-37.79, 158.48, 59.84) mm, rotated rx 180 ry 0 rz 180 deg; joints [-53.226, -12.612, 82.591, 75.647, 55.772, -65.539]
  MoveL 3154 to (-37.79, 158.48, 59.84) mm, rotated rx 180 ry 0 rz 180 deg; joints [-53.226, -12.612, 82.591, 75.647, 55.772, -65.539]
  Call Extruder(7.01744)
  MoveL 3155 to (-38.12, 158.02, 59.84) mm, rotated rx -180 ry 0 rz -180 deg; joints [-53.224, -12.69, 82.651, 75.635, 55.775, -65.517]
  MoveL 3156 to (-38.12, 158.02, 59.84) mm, rotated rx -180 ry 0 rz -180 deg; joints [-53.224, -12.69, 82.651, 75.635, 55.775, -65.517]
  Call Extruder(7.13511)
  MoveL 3157 to (-38.22, 157.85, 59.84) mm, rotated rx 180 ry 0 rz 180 deg; joints [-53.221, -12.718, 82.673, 75.629, 55.773, -65.509]
  MoveL 3158 to (-38.22, 157.85, 59.84) mm, rotated rx 180 ry 0 rz 180 deg; joints [-53.221, -12.718, 82.673, 75.629, 55.773, -65.509]
  Call Extruder(7.34283)
  MoveL 3159 to (-38.4, 157.55, 59.84) mm, rotated rx 180 ry 0 rz 180 deg; joints [-53.214, -12.767, 82.71, 75.618, 55.77, -65.494]
  MoveL 3160 to (-38.4, 157.55, 59.84) mm, rotated rx 180 ry 0 rz 180 deg; joints [-53.214, -12.767, 82.71, 75.618, 55.77, -65.494]
  Call Extruder(7.54978)
  MoveL 3161 to (-38.57, 157.25, 59.84) mm, rotated rx 180 ry 0 rz 180 deg; joints [-53.207, -12.816, 82.748, 75.607, 55.766, -65.478]
  MoveL 3162 to (-38.57, 157.25, 59.84) mm, rotated rx 180 ry 0 rz 180 deg; joints [-53.207, -12.816, 82.748, 75.607, 55.766, -65.478]
  Call Extruder(7.75595)
  MoveL 3163 to (-38.75, 156.94, 59.84) mm, rotated rx 180 ry 0 rz 180 deg; joints [-53.2, -12.865, 82.786, 75.596, 55.763, -65.463]
  MoveL 3164 to (-38.75, 156.94, 59.84) mm, rotated rx 180 ry 0 rz 180 deg; joints [-53.2, -12.865, 82.786, 75.596, 55.763, -65.463]
  Call Extruder(7.93763)
  MoveL 3165 to (-38.89, 156.66, 59.84) mm, rotated rx 180 ry 0 rz -180 deg; joints [-53.191, -12.908, 82.819, 75.585, 55.757, -65.449]
  MoveL 3166 to (-38.89, 156.66, 59.84) mm, rotated rx 180 ry 0 rz -180 deg; joints [-53.191, -12.908, 82.819, 75.585, 55.757, -65.449]
  Call Extruder(8.09561)
  MoveL 3167 to (-39, 156.42, 59.84) mm, rotated rx 180 ry 0 rz 180 deg; joints [-53.18, -12.945, 82.847, 75.574, 55.75, -65.436]
  MoveL 3168 to (-39, 156.42, 59.84) mm, rotated rx 180 ry 0 rz 180 deg; joints [-53.18, -12.945, 82.847, 75.574, 55.75, -65.436]
  Call Extruder(8.25300)
  MoveL 3169 to (-39.11, 156.17, 59.84) mm, rotated rx -180 ry 0 rz 180 deg; joints [-53.17, -12.982, 82.875, 75.563, 55.742, -65.423]
  MoveL 3170 to (-39.11, 156.17, 59.84) mm, rotated rx -180 ry 0 rz 180 deg; joints [-53.17, -12.982, 82.875, 75.563, 55.742, -65.423]
  Call Extruder(8.43572)
  MoveL 3171 to (-39.22, 155.88, 59.84) mm, rotated rx 180 ry 0 rz 180 deg; joints [-53.156, -13.025, 82.908, 75.549, 55.733, -65.407]
  MoveL 3172 to (-39.22, 155.88, 59.84) mm, rotated rx 180 ry 0 rz 180 deg; joints [-53.156, -13.025, 82.908, 75.549, 55.733, -65.407]
  Call Extruder(8.61768)
  MoveL 3173 to (-39.35, 155.58, 59.84) mm, rotated rx 180 ry 0 rz 180 deg; joints [-53.143, -13.068, 82.941, 75.536, 55.724, -65.391]
  MoveL 3174 to (-39.35, 155.58, 59.84) mm, rotated rx 180 ry 0 rz 180 deg; joints [-53.143, -13.068, 82.941, 75.536, 55.724, -65.391]
  Call Extruder(8.76501)
  MoveL 3175 to (-39.44, 155.34, 59.84) mm, rotated rx -180 ry 0 rz 180 deg; joints [-53.131, -13.102, 82.967, 75.525, 55.715, -65.379]
  MoveL 3176 to (-39.44, 155.34, 59.84) mm, rotated rx -180 ry 0 rz 180 deg; joints [-53.131, -13.102, 82.967, 75.525, 55.715, -65.379]
  Call Extruder(8.87825)
  MoveL 3177 to (-39.5, 155.15, 59.84) mm, rotated rx 180 ry 0 rz 180 deg; joints [-53.121, -13.129, 82.988, 75.515, 55.707, -65.368]
  MoveL 3178 to (-39.5, 155.15, 59.84) mm, rotated rx 180 ry 0 rz 180 deg; joints [-53.121, -13.129, 82.988, 75.515, 55.707, -65.368]
  Call Extruder(8.99104)
  MoveL 3179 to (-39.56, 154.97, 59.84) mm, rotated rx -180 ry 0 rz 180 deg; joints [-53.11, -13.155, 83.008, 75.505, 55.698, -65.358]
  MoveL 3180 to (-39.56, 154.97, 59.84) mm, rotated rx -180 ry 0 rz 180 deg; joints [-53.11, -13.155, 83.008, 75.505, 55.698, -65.358]
  Call Extruder(9.10338)
  MoveL 3181 to (-39.62, 154.78, 59.84) mm, rotated rx 180 ry 0 rz 180 deg; joints [-53.099, -13.181, 83.028, 75.496, 55.69, -65.347]
  MoveL 3182 to (-39.62, 154.78, 59.84) mm, rotated rx 180 ry 0 rz 180 deg; joints [-53.099, -13.181, 83.028, 75.496, 55.69, -65.347]
  Call Extruder(9.21528)
  MoveL 3183 to (-39.68, 154.59, 59.84) mm, rotated rx -180 ry 0 rz -180 deg; joints [-53.088, -13.208, 83.048, 75.486, 55.682, -65.337]
  MoveL 3184 to (-39.68, 154.59, 59.84) mm, rotated rx -180 ry 0 rz -180 deg; joints [-53.088, -13.208, 83.048, 75.486, 55.682, -65.337]
  Call Extruder(9.33668)
  MoveL 3185 to (-39.75, 154.38, 59.84) mm, rotated rx 180 ry 0 rz -180 deg; joints [-53.076, -13.236, 83.069, 75.476, 55.673, -65.325]
  MoveL 3186 to (-39.75, 154.38, 59.84) mm, rotated rx 180 ry 0 rz -180 deg; joints [-53.076, -13.236, 83.069, 75.476, 55.673, -65.325]
  Call Extruder(9.46748)
  MoveL 3187 to (-39.81, 154.16, 59.84) mm, rotated rx 180 ry 0 rz 180 deg; joints [-53.063, -13.267, 83.093, 75.464, 55.662, -65.313]
  MoveL 3188 to (-39.81, 154.16, 59.84) mm, rotated rx 180 ry 0 rz 180 deg; joints [-53.063, -13.267, 83.093, 75.464, 55.662, -65.313]
  Call Extruder(9.59771)
  MoveL 3189 to (-39.88, 153.94, 59.84) mm, rotated rx 180 ry 0 rz 180 deg; joints [-53.049, -13.297, 83.116, 75.452, 55.652, -65.3]
  MoveL 3190 to (-39.88, 153.94, 59.84) mm, rotated rx 180 ry 0 rz 180 deg; joints [-53.049, -13.297, 83.116, 75.452, 55.652, -65.3]
  Call Extruder(9.72737)
  MoveL 3191 to (-39.95, 153.71, 59.84) mm, rotated rx 180 ry 0 rz -180 deg; joints [-53.036, -13.328, 83.139, 75.44, 55.641, -65.288]
  MoveL 3192 to (-39.95, 153.71, 59.84) mm, rotated rx 180 ry 0 rz -180 deg; joints [-53.036, -13.328, 83.139, 75.44, 55.641, -65.288]
  Call Extruder(9.85647)
  MoveL 3193 to (-40.02, 153.49, 59.84) mm, rotated rx -180 ry 0 rz 180 deg; joints [-53.022, -13.359, 83.163, 75.429, 55.631, -65.275]
  MoveL 3194 to (-40.02, 153.49, 59.84) mm, rotated rx -180 ry 0 rz 180 deg; joints [-53.022, -13.359, 83.163, 75.429, 55.631, -65.275]
  Call Extruder(9.97156)
  MoveL 3195 to (-40.06, 153.28, 59.84) mm, rotated rx 180 ry 0 rz 180 deg; joints [-53.007, -13.386, 83.183, 75.417, 55.619, -65.264]
  MoveL 3196 to (-40.06, 153.28, 59.84) mm, rotated rx 180 ry 0 rz 180 deg; joints [-53.007, -13.386, 83.183, 75.417, 55.619, -65.264]
  Call Extruder(10.08619)
  MoveL 3197 to (-40.11, 153.08, 59.84) mm, rotated rx -180 ry 0 rz 180 deg; joints [-52.993, -13.412, 83.203, 75.405, 55.607, -65.252]
  MoveL 3198 to (-40.11, 153.08, 59.84) mm, rotated rx -180 ry 0 rz 180 deg; joints [-52.993, -13.412, 83.203, 75.405, 55.607, -65.252]
  Call Extruder(10.20037)
  MoveL 3199 to (-40.15, 152.88, 59.84) mm, rotated rx 180 ry 0 rz 180 deg; joints [-52.978, -13.439, 83.223, 75.393, 55.595, -65.24]
  MoveL 3200 to (-40.15, 152.88, 59.84) mm, rotated rx 180 ry 0 rz 180 deg; joints [-52.978, -13.439, 83.223, 75.393, 55.595, -65.24]
  Call Extruder(10.31410)
  MoveL 3201 to (-40.2, 152.67, 59.84) mm, rotated rx 180 ry 0 rz 180 deg; joints [-52.963, -13.465, 83.243, 75.382, 55.584, -65.228]
  MoveL 3202 to (-40.2, 152.67, 59.84) mm, rotated rx 180 ry 0 rz 180 deg; joints [-52.963, -13.465, 83.243, 75.382, 55.584, -65.228]
  Call Extruder(10.43953)
  MoveL 3203 to (-40.24, 152.45, 59.84) mm, rotated rx -180 ry 0 rz -180 deg; joints [-52.946, -13.494, 83.265, 75.368, 55.57, -65.215]
  MoveL 3204 to (-40.24, 152.45, 59.84) mm, rotated rx -180 ry 0 rz -180 deg; joints [-52.946, -13.494, 83.265, 75.368, 55.57, -65.215]
  Call Extruder(10.57650)
  MoveL 3205 to (-40.29, 152.2, 59.84) mm, rotated rx 180 ry 0 rz 180 deg; joints [-52.928, -13.526, 83.29, 75.354, 55.555, -65.201]
  MoveL 3206 to (-40.29, 152.2, 59.84) mm, rotated rx 180 ry 0 rz 180 deg; joints [-52.928, -13.526, 83.29, 75.354, 55.555, -65.201]
  Call Extruder(10.71287)
  MoveL 3207 to (-40.34, 151.95, 59.84) mm, rotated rx 180 ry 0 rz 180 deg; joints [-52.909, -13.559, 83.314, 75.339, 55.54, -65.186]
  MoveL 3208 to (-40.34, 151.95, 59.84) mm, rotated rx 180 ry 0 rz 180 deg; joints [-52.909, -13.559, 83.314, 75.339, 55.54, -65.186]
  Call Extruder(10.84862)
  MoveL 3209 to (-40.39, 151.7, 59.84) mm, rotated rx -180 ry 0 rz 180 deg; joints [-52.89, -13.59, 83.338, 75.324, 55.525, -65.171]
  MoveL 3210 to (-40.39, 151.7, 59.84) mm, rotated rx -180 ry 0 rz 180 deg; joints [-52.89, -13.59, 83.338, 75.324, 55.525, -65.171]
  Call Extruder(10.98377)
  MoveL 3211 to (-40.44, 151.45, 59.84) mm, rotated rx 180 ry 0 rz 180 deg; joints [-52.871, -13.622, 83.362, 75.309, 55.51, -65.157]
  MoveL 3212 to (-40.44, 151.45, 59.84) mm, rotated rx 180 ry 0 rz 180 deg; joints [-52.871, -13.622, 83.362, 75.309, 55.51, -65.157]
  Call Extruder(11.11831)
  MoveL 3213 to (-40.49, 151.2, 59.84) mm, rotated rx -180 ry 0 rz 180 deg; joints [-52.853, -13.654, 83.386, 75.295, 55.495, -65.142]
  MoveL 3214 to (-40.49, 151.2, 59.84) mm, rotated rx -180 ry 0 rz 180 deg; joints [-52.853, -13.654, 83.386, 75.295, 55.495, -65.142]
  Call Extruder(11.25223)
  MoveL 3215 to (-40.54, 150.95, 59.84) mm, rotated rx 180 ry 0 rz 180 deg; joints [-52.834, -13.686, 83.41, 75.28, 55.48, -65.127]
  MoveL 3216 to (-40.54, 150.95, 59.84) mm, rotated rx 180 ry 0 rz 180 deg; joints [-52.834, -13.686, 83.41, 75.28, 55.48, -65.127]
  Call Extruder(11.40009)
  MoveL 3217 to (-40.59, 150.67, 59.84) mm, rotated rx -180 ry 0 rz 180 deg; joints [-52.812, -13.721, 83.436, 75.263, 55.462, -65.111]
  MoveL 3218 to (-40.59, 150.67, 59.84) mm, rotated rx -180 ry 0 rz 180 deg; joints [-52.812, -13.721, 83.436, 75.263, 55.462, -65.111]
  Call Extruder(11.56181)
  MoveL 3219 to (-40.64, 150.37, 59.84) mm, rotated rx 180 ry 0 rz 180 deg; joints [-52.787, -13.759, 83.465, 75.244, 55.442, -65.092]
  MoveL 3220 to (-40.64, 150.37, 59.84) mm, rotated rx 180 ry 0 rz 180 deg; joints [-52.787, -13.759, 83.465, 75.244, 55.442, -65.092]
  Call Extruder(11.72281)
  MoveL 3221 to (-40.69, 150.06, 59.84) mm, rotated rx 180 ry 0 rz 180 deg; joints [-52.762, -13.797, 83.493, 75.225, 55.422, -65.074]
  MoveL 3222 to (-40.69, 150.06, 59.84) mm, rotated rx 180 ry 0 rz 180 deg; joints [-52.762, -13.797, 83.493, 75.225, 55.422, -65.074]
  Call Extruder(11.88308)
  MoveL 3223 to (-40.73, 149.76, 59.84) mm, rotated rx 180 ry 0 rz 180 deg; joints [-52.737, -13.835, 83.522, 75.206, 55.402, -65.056]
  MoveL 3224 to (-40.73, 149.76, 59.84) mm, rotated rx 180 ry 0 rz 180 deg; joints [-52.737, -13.835, 83.522, 75.206, 55.402, -65.056]
  Call Extruder(12.04262)
  MoveL 3225 to (-40.78, 149.45, 59.84) mm, rotated rx 180 ry 0 rz -180 deg; joints [-52.712, -13.873, 83.55, 75.186, 55.382, -65.037]
  MoveL 3226 to (-40.78, 149.45, 59.84) mm, rotated rx 180 ry 0 rz -180 deg; joints [-52.712, -13.873, 83.55, 75.186, 55.382, -65.037]
  Call Extruder(12.20144)
  MoveL 3227 to (-40.83, 149.14, 59.84) mm, rotated rx 180 ry 0 rz 180 deg; joints [-52.687, -13.911, 83.579, 75.167, 55.361, -65.019]
  MoveL 3228 to (-40.83, 149.14, 59.84) mm, rotated rx 180 ry 0 rz 180 deg; joints [-52.687, -13.911, 83.579, 75.167, 55.361, -65.019]
  Call Extruder(12.38010)
  MoveL 3229 to (-40.88, 148.8, 59.84) mm, rotated rx -180 ry 0 rz 180 deg; joints [-52.658, -13.954, 83.611, 75.145, 55.337, -64.997]
  MoveL 3230 to (-40.88, 148.8, 59.84) mm, rotated rx -180 ry 0 rz 180 deg; joints [-52.658, -13.954, 83.611, 75.145, 55.337, -64.997]
  Call Extruder(12.57854)
  MoveL 3231 to (-40.93, 148.41, 59.84) mm, rotated rx -180 ry 0 rz 180 deg; joints [-52.624, -14.001, 83.646, 75.12, 55.31, -64.974]
  MoveL 3232 to (-40.93, 148.41, 59.84) mm, rotated rx -180 ry 0 rz 180 deg; joints [-52.624, -14.001, 83.646, 75.12, 55.31, -64.974]
  Call Extruder(12.77612)
  MoveL 3233 to (-40.97, 148.02, 59.84) mm, rotated rx -180 ry 0 rz 180 deg; joints [-52.59, -14.047, 83.68, 75.094, 55.282, -64.95]
  MoveL 3234 to (-40.97, 148.02, 59.84) mm, rotated rx -180 ry 0 rz 180 deg; joints [-52.59, -14.047, 83.68, 75.094, 55.282, -64.95]
  Call Extruder(12.97282)
  MoveL 3235 to (-41.02, 147.63, 59.84) mm, rotated rx -180 ry 0 rz -180 deg; joints [-52.556, -14.094, 83.715, 75.069, 55.254, -64.926]
  MoveL 3236 to (-41.02, 147.63, 59.84) mm, rotated rx -180 ry 0 rz -180 deg; joints [-52.556, -14.094, 83.715, 75.069, 55.254, -64.926]
  Call Extruder(13.16866)
  MoveL 3237 to (-41.06, 147.25, 59.84) mm, rotated rx 180 ry 0 rz -180 deg; joints [-52.521, -14.141, 83.75, 75.043, 55.226, -64.902]
  MoveL 3238 to (-41.06, 147.25, 59.84) mm, rotated rx 180 ry 0 rz -180 deg; joints [-52.521, -14.141, 83.75, 75.043, 55.226, -64.902]
  Call Extruder(13.46406)
  MoveL 3239 to (-41.11, 146.66, 59.84) mm, rotated rx -180 ry 0 rz 180 deg; joints [-52.466, -14.21, 83.801, 75.002, 55.181, -64.864]
  MoveL 3240 to (-41.11, 146.66, 59.84) mm, rotated rx -180 ry 0 rz 180 deg; joints [-52.466, -14.21, 83.801, 75.002, 55.181, -64.864]
  Call Extruder(13.75812)
  MoveL 3241 to (-41.16, 146.07, 59.84) mm, rotated rx 180 ry 0 rz 180 deg; joints [-52.411, -14.279, 83.852, 74.962, 55.135, -64.827]
  MoveL 3242 to (-41.16, 146.07, 59.84) mm, rotated rx 180 ry 0 rz 180 deg; joints [-52.411, -14.279, 83.852, 74.962, 55.135, -64.827]
  Call Extruder(14.05086)
  MoveL 3243 to (-41.2, 145.48, 59.84) mm, rotated rx 180 ry 0 rz 180 deg; joints [-52.355, -14.348, 83.903, 74.921, 55.09, -64.79]
  MoveL 3244 to (-41.2, 145.48, 59.84) mm, rotated rx 180 ry 0 rz 180 deg; joints [-52.355, -14.348, 83.903, 74.921, 55.09, -64.79]
  Call Extruder(14.62431)
  MoveL 3245 to (-41.25, 144.32, 59.84) mm, rotated rx 180 ry 0 rz 180 deg; joints [-52.239, -14.479, 84.001, 74.837, 54.993, -64.714]
  MoveL 3246 to (-41.25, 144.32, 59.84) mm, rotated rx 180 ry 0 rz 180 deg; joints [-52.239, -14.479, 84.001, 74.837, 54.993, -64.714]
  Call Extruder(15.33827)
  MoveL 3247 to (-41.29, 142.86, 59.84) mm, rotated rx -180 ry 0 rz 180 deg; joints [-52.09, -14.642, 84.121, 74.73, 54.87, -64.619]
  Call Extruder(57.40310)
  MoveL 3248 to (-41.29, 57.14, 59.84) mm, rotated rx -180 ry 0 rz 180 deg; joints [-40.759, -23.035, 89.623, 65.251, 45.964, -56.448]
  Call Extruder(57.83165)
  MoveL 3249 to (-41.27, 56.26, 59.84) mm, rotated rx 180 ry 0 rz 180 deg; joints [-40.614, -23.107, 89.664, 65.112, 45.857, -56.331]
  MoveL 3250 to (-41.27, 56.26, 59.84) mm, rotated rx 180 ry 0 rz 180 deg; joints [-40.614, -23.107, 89.664, 65.112, 45.857, -56.331]
  Call Extruder(58.11773)
  MoveL 3251 to (-41.25, 55.68, 59.84) mm, rotated rx 180 ry 0 rz 180 deg; joints [-40.517, -23.154, 89.691, 65.019, 45.784, -56.253]
  MoveL 3252 to (-41.25, 55.68, 59.84) mm, rotated rx 180 ry 0 rz 180 deg; joints [-40.517, -23.154, 89.691, 65.019, 45.784, -56.253]
  Call Extruder(58.69247)
  MoveL 3253 to (-41.2, 54.52, 59.84) mm, rotated rx 180 ry 0 rz 180 deg; joints [-40.32, -23.248, 89.745, 64.831, 45.638, -56.096]
  MoveL 3254 to (-41.2, 54.52, 59.84) mm, rotated rx 180 ry 0 rz 180 deg; joints [-40.32, -23.248, 89.745, 64.831, 45.638, -56.096]
  Call Extruder(58.98587)
  MoveL 3255 to (-41.15, 53.93, 59.84) mm, rotated rx -180 ry 0 rz 180 deg; joints [-40.217, -23.293, 89.77, 64.733, 45.561, -56.015]
  MoveL 3256 to (-41.15, 53.93, 59.84) mm, rotated rx -180 ry 0 rz 180 deg; joints [-40.217, -23.293, 89.77, 64.733, 45.561, -56.015]
  Call Extruder(59.28060)
  MoveL 3257 to (-41.11, 53.34, 59.84) mm, rotated rx 180 ry 0 rz 180 deg; joints [-40.114, -23.338, 89.796, 64.635, 45.483, -55.933]
  MoveL 3258 to (-41.11, 53.34, 59.84) mm, rotated rx 180 ry 0 rz 180 deg; joints [-40.114, -23.338, 89.796, 64.635, 45.483, -55.933]
  Call Extruder(59.57666)
  MoveL 3259 to (-41.06, 52.75, 59.84) mm, rotated rx 180 ry 0 rz 180 deg; joints [-40.01, -23.382, 89.821, 64.536, 45.406, -55.852]
  MoveL 3260 to (-41.06, 52.75, 59.84) mm, rotated rx 180 ry 0 rz 180 deg; joints [-40.01, -23.382, 89.821, 64.536, 45.406, -55.852]
  Call Extruder(59.77294)
  MoveL 3261 to (-41.02, 52.36, 59.84) mm, rotated rx 180 ry 0 rz 180 deg; joints [-39.939, -23.41, 89.837, 64.469, 45.353, -55.797]
  MoveL 3262 to (-41.02, 52.36, 59.84) mm, rotated rx 180 ry 0 rz 180 deg; joints [-39.939, -23.41, 89.837, 64.469, 45.353, -55.797]
  Call Extruder(59.97008)
  MoveL 3263 to (-40.97, 51.98, 59.84) mm, rotated rx 180 ry 0 rz 180 deg; joints [-39.869, -23.438, 89.853, 64.403, 45.299, -55.743]
  MoveL 3264 to (-40.97, 51.98, 59.84) mm, rotated rx 180 ry 0 rz 180 deg; joints [-39.869, -23.438, 89.853, 64.403, 45.299, -55.743]
  Call Extruder(60.16808)
  MoveL 3265 to (-40.92, 51.59, 59.84) mm, rotated rx 180 ry 0 rz 180 deg; joints [-39.798, -23.466, 89.869, 64.336, 45.246, -55.688]
  MoveL 3266 to (-40.92, 51.59, 59.84) mm, rotated rx 180 ry 0 rz 180 deg; joints [-39.798, -23.466, 89.869, 64.336, 45.246, -55.688]
  Call Extruder(60.36696)
  MoveL 3267 to (-40.88, 51.2, 59.84) mm, rotated rx -180 ry 0 rz 180 deg; joints [-39.727, -23.493, 89.884, 64.269, 45.193, -55.633]
  MoveL 3268 to (-40.88, 51.2, 59.84) mm, rotated rx -180 ry 0 rz 180 deg; joints [-39.727, -23.493, 89.884, 64.269, 45.193, -55.633]
  Call Extruder(60.54604)
  MoveL 3269 to (-40.83, 50.86, 59.84) mm, rotated rx -180 ry 0 rz 180 deg; joints [-39.663, -23.517, 89.898, 64.209, 45.144, -55.584]
  MoveL 3270 to (-40.83, 50.86, 59.84) mm, rotated rx -180 ry 0 rz 180 deg; joints [-39.663, -23.517, 89.898, 64.209, 45.144, -55.584]
  Call Extruder(60.70522)
  MoveL 3271 to (-40.78, 50.55, 59.84) mm, rotated rx 180 ry 0 rz 180 deg; joints [-39.605, -23.538, 89.909, 64.154, 45.1, -55.54]
  MoveL 3272 to (-40.78, 50.55, 59.84) mm, rotated rx 180 ry 0 rz 180 deg; joints [-39.605, -23.538, 89.909, 64.154, 45.1, -55.54]
  Call Extruder(60.86512)
  MoveL 3273 to (-40.74, 50.24, 59.84) mm, rotated rx 180 ry 0 rz 180 deg; joints [-39.547, -23.558, 89.921, 64.1, 45.057, -55.496]
  MoveL 3274 to (-40.74, 50.24, 59.84) mm, rotated rx 180 ry 0 rz 180 deg; joints [-39.547, -23.558, 89.921, 64.1, 45.057, -55.496]
  Call Extruder(61.02576)
  MoveL 3275 to (-40.69, 49.94, 59.84) mm, rotated rx 180 ry 0 rz 180 deg; joints [-39.489, -23.579, 89.932, 64.046, 45.013, -55.452]
  MoveL 3276 to (-40.69, 49.94, 59.84) mm, rotated rx 180 ry 0 rz 180 deg; joints [-39.489, -23.579, 89.932, 64.046, 45.013, -55.452]
  Call Extruder(61.18712)
  MoveL 3277 to (-40.64, 49.63, 59.84) mm, rotated rx 180 ry 0 rz 180 deg; joints [-39.431, -23.599, 89.944, 63.991, 44.969, -55.408]
  MoveL 3278 to (-40.64, 49.63, 59.84) mm, rotated rx 180 ry 0 rz 180 deg; joints [-39.431, -23.599, 89.944, 63.991, 44.969, -55.408]
  Call Extruder(61.34921)
  MoveL 3279 to (-40.59, 49.33, 59.84) mm, rotated rx 180 ry 0 rz 180 deg; joints [-39.373, -23.619, 89.955, 63.937, 44.925, -55.364]
  MoveL 3280 to (-40.59, 49.33, 59.84) mm, rotated rx 180 ry 0 rz 180 deg; joints [-39.373, -23.619, 89.955, 63.937, 44.925, -55.364]
  Call Extruder(61.49741)
  MoveL 3281 to (-40.54, 49.05, 59.84) mm, rotated rx -180 ry 0 rz 180 deg; joints [-39.32, -23.637, 89.965, 63.887, 44.885, -55.323]
  MoveL 3282 to (-40.54, 49.05, 59.84) mm, rotated rx -180 ry 0 rz 180 deg; joints [-39.32, -23.637, 89.965, 63.887, 44.885, -55.323]
  Call Extruder(61.63164)
  MoveL 3283 to (-40.49, 48.8, 59.84) mm, rotated rx 180 ry 0 rz 180 deg; joints [-39.271, -23.653, 89.974, 63.841, 44.848, -55.287]
  MoveL 3284 to (-40.49, 48.8, 59.84) mm, rotated rx 180 ry 0 rz 180 deg; joints [-39.271, -23.653, 89.974, 63.841, 44.848, -55.287]
  Call Extruder(61.76648)
  MoveL 3285 to (-40.44, 48.55, 59.84) mm, rotated rx 180 ry 0 rz 180 deg; joints [-39.222, -23.668, 89.983, 63.796, 44.811, -55.25]
  MoveL 3286 to (-40.44, 48.55, 59.84) mm, rotated rx 180 ry 0 rz 180 deg; joints [-39.222, -23.668, 89.983, 63.796, 44.811, -55.25]
  Call Extruder(61.90193)
  MoveL 3287 to (-40.39, 48.3, 59.84) mm, rotated rx -180 ry 0 rz 180 deg; joints [-39.174, -23.684, 89.992, 63.75, 44.774, -55.213]
  MoveL 3288 to (-40.39, 48.3, 59.84) mm, rotated rx -180 ry 0 rz 180 deg; joints [-39.174, -23.684, 89.992, 63.75, 44.774, -55.213]
  Call Extruder(62.03799)
  MoveL 3289 to (-40.34, 48.05, 59.84) mm, rotated rx 180 ry 0 rz 180 deg; joints [-39.125, -23.699, 90, 63.704, 44.736, -55.177]
  MoveL 3290 to (-40.34, 48.05, 59.84) mm, rotated rx 180 ry 0 rz 180 deg; joints [-39.125, -23.699, 90, 63.704, 44.736, -55.177]
  Call Extruder(62.17466)
  MoveL 3291 to (-40.29, 47.8, 59.84) mm, rotated rx -180 ry 0 rz -180 deg; joints [-39.076, -23.714, 90.009, 63.658, 44.699, -55.14]
  MoveL 3292 to (-40.29, 47.8, 59.84) mm, rotated rx -180 ry 0 rz -180 deg; joints [-39.076, -23.714, 90.009, 63.658, 44.699, -55.14]
  Call Extruder(62.31194)
  MoveL 3293 to (-40.24, 47.56, 59.84) mm, rotated rx -180 ry 0 rz 180 deg; joints [-39.027, -23.73, 90.017, 63.612, 44.662, -55.103]
  MoveL 3294 to (-40.24, 47.56, 59.84) mm, rotated rx -180 ry 0 rz 180 deg; joints [-39.027, -23.73, 90.017, 63.612, 44.662, -55.103]
  Call Extruder(62.43761)
  MoveL 3295 to (-40.2, 47.33, 59.84) mm, rotated rx 180 ry 0 rz 180 deg; joints [-38.982, -23.743, 90.025, 63.571, 44.628, -55.069]
  MoveL 3296 to (-40.2, 47.33, 59.84) mm, rotated rx 180 ry 0 rz 180 deg; joints [-38.982, -23.743, 90.025, 63.571, 44.628, -55.069]
  Call Extruder(62.55157)
  MoveL 3297 to (-40.15, 47.12, 59.84) mm, rotated rx -180 ry 0 rz 180 deg; joints [-38.941, -23.756, 90.032, 63.532, 44.597, -55.039]
  MoveL 3298 to (-40.15, 47.12, 59.84) mm, rotated rx -180 ry 0 rz 180 deg; joints [-38.941, -23.756, 90.032, 63.532, 44.597, -55.039]
  Call Extruder(62.66597)
  MoveL 3299 to (-40.11, 46.92, 59.84) mm, rotated rx 180 ry 0 rz -180 deg; joints [-38.9, -23.768, 90.039, 63.494, 44.566, -55.008]
  MoveL 3300 to (-40.11, 46.92, 59.84) mm, rotated rx 180 ry 0 rz -180 deg; joints [-38.9, -23.768, 90.039, 63.494, 44.566, -55.008]
  Call Extruder(62.78083)
  MoveL 3301 to (-40.06, 46.72, 59.84) mm, rotated rx -180 ry 0 rz 180 deg; joints [-38.859, -23.78, 90.046, 63.456, 44.535, -54.978]
  MoveL 3302 to (-40.06, 46.72, 59.84) mm, rotated rx -180 ry 0 rz 180 deg; joints [-38.859, -23.78, 90.046, 63.456, 44.535, -54.978]
  Call Extruder(62.89615)
  MoveL 3303 to (-40.02, 46.51, 59.84) mm, rotated rx -180 ry 0 rz 180 deg; joints [-38.819, -23.792, 90.052, 63.418, 44.504, -54.947]
  MoveL 3304 to (-40.02, 46.51, 59.84) mm, rotated rx -180 ry 0 rz 180 deg; joints [-38.819, -23.792, 90.052, 63.418, 44.504, -54.947]
  Call Extruder(63.02553)
  MoveL 3305 to (-39.95, 46.29, 59.84) mm, rotated rx -180 ry 0 rz 180 deg; joints [-38.771, -23.803, 90.059, 63.374, 44.467, -54.913]
  MoveL 3306 to (-39.95, 46.29, 59.84) mm, rotated rx -180 ry 0 rz 180 deg; joints [-38.771, -23.803, 90.059, 63.374, 44.467, -54.913]
  Call Extruder(63.15547)
  MoveL 3307 to (-39.88, 46.06, 59.84) mm, rotated rx 180 ry 0 rz 180 deg; joints [-38.724, -23.815, 90.065, 63.331, 44.43, -54.879]
  MoveL 3308 to (-39.88, 46.06, 59.84) mm, rotated rx 180 ry 0 rz 180 deg; joints [-38.724, -23.815, 90.065, 63.331, 44.43, -54.879]
  Call Extruder(63.28598)
  MoveL 3309 to (-39.82, 45.84, 59.84) mm, rotated rx 180 ry 0 rz 180 deg; joints [-38.677, -23.826, 90.071, 63.287, 44.394, -54.845]
  MoveL 3310 to (-39.82, 45.84, 59.84) mm, rotated rx 180 ry 0 rz 180 deg; joints [-38.677, -23.826, 90.071, 63.287, 44.394, -54.845]
  Call Extruder(63.41706)
  MoveL 3311 to (-39.75, 45.62, 59.84) mm, rotated rx 180 ry 0 rz 180 deg; joints [-38.629, -23.837, 90.078, 63.244, 44.357, -54.81]
  MoveL 3312 to (-39.75, 45.62, 59.84) mm, rotated rx 180 ry 0 rz 180 deg; joints [-38.629, -23.837, 90.078, 63.244, 44.357, -54.81]
  Call Extruder(63.53870)
  MoveL 3313 to (-39.68, 45.41, 59.84) mm, rotated rx 180 ry 0 rz 180 deg; joints [-38.585, -23.847, 90.083, 63.203, 44.323, -54.779]
  MoveL 3314 to (-39.68, 45.41, 59.84) mm, rotated rx 180 ry 0 rz 180 deg; joints [-38.585, -23.847, 90.083, 63.203, 44.323, -54.779]
  Call Extruder(63.65083)
  MoveL 3315 to (-39.62, 45.22, 59.84) mm, rotated rx 180 ry 0 rz 180 deg; joints [-38.544, -23.856, 90.088, 63.166, 44.292, -54.75]
  MoveL 3316 to (-39.62, 45.22, 59.84) mm, rotated rx 180 ry 0 rz 180 deg; joints [-38.544, -23.856, 90.088, 63.166, 44.292, -54.75]
  Call Extruder(63.76340)
  MoveL 3317 to (-39.56, 45.03, 59.84) mm, rotated rx 180 ry 0 rz 180 deg; joints [-38.504, -23.865, 90.093, 63.129, 44.261, -54.72]
  MoveL 3318 to (-39.56, 45.03, 59.84) mm, rotated rx 180 ry 0 rz 180 deg; joints [-38.504, -23.865, 90.093, 63.129, 44.261, -54.72]
  Call Extruder(63.87641)
  MoveL 3319 to (-39.5, 44.85, 59.84) mm, rotated rx 180 ry 0 rz 180 deg; joints [-38.463, -23.874, 90.098, 63.092, 44.229, -54.691]
  MoveL 3320 to (-39.5, 44.85, 59.84) mm, rotated rx 180 ry 0 rz 180 deg; joints [-38.463, -23.874, 90.098, 63.092, 44.229, -54.691]
  Call Extruder(63.98987)
  MoveL 3321 to (-39.44, 44.66, 59.84) mm, rotated rx 180 ry 0 rz 180 deg; joints [-38.422, -23.883, 90.103, 63.054, 44.198, -54.662]
  MoveL 3322 to (-39.44, 44.66, 59.84) mm, rotated rx 180 ry 0 rz 180 deg; joints [-38.422, -23.883, 90.103, 63.054, 44.198, -54.662]
  Call Extruder(64.13751)
  MoveL 3323 to (-39.35, 44.42, 59.84) mm, rotated rx 180 ry 0 rz 180 deg; joints [-38.369, -23.893, 90.109, 63.006, 44.156, -54.624]
  MoveL 3324 to (-39.35, 44.42, 59.84) mm, rotated rx 180 ry 0 rz 180 deg; joints [-38.369, -23.893, 90.109, 63.006, 44.156, -54.624]
  Call Extruder(64.31985)
  MoveL 3325 to (-39.22, 44.13, 59.84) mm, rotated rx 180 ry 0 rz 180 deg; joints [-38.302, -23.904, 90.115, 62.946, 44.104, -54.578]
  MoveL 3326 to (-39.22, 44.13, 59.84) mm, rotated rx 180 ry 0 rz 180 deg; joints [-38.302, -23.904, 90.115, 62.946, 44.104, -54.578]
  Call Extruder(64.50294)
  MoveL 3327 to (-39.11, 43.83, 59.84) mm, rotated rx 180 ry 0 rz 180 deg; joints [-38.236, -23.916, 90.121, 62.886, 44.052, -54.532]
  MoveL 3328 to (-39.11, 43.83, 59.84) mm, rotated rx 180 ry 0 rz 180 deg; joints [-38.236, -23.916, 90.121, 62.886, 44.052, -54.532]
  Call Extruder(64.66063)
  MoveL 3329 to (-39, 43.58, 59.84) mm, rotated rx 180 ry 0 rz 180 deg; joints [-38.178, -23.925, 90.126, 62.834, 44.007, -54.492]
  MoveL 3330 to (-39, 43.58, 59.84) mm, rotated rx 180 ry 0 rz 180 deg; joints [-38.178, -23.925, 90.126, 62.834, 44.007, -54.492]
  Call Extruder(64.81891)
  MoveL 3331 to (-38.89, 43.33, 59.84) mm, rotated rx -180 ry 0 rz 180 deg; joints [-38.121, -23.934, 90.131, 62.782, 43.962, -54.453]
  MoveL 3332 to (-38.89, 43.33, 59.84) mm, rotated rx -180 ry 0 rz 180 deg; joints [-38.121, -23.934, 90.131, 62.782, 43.962, -54.453]
  Call Extruder(65.00094)
  MoveL 3333 to (-38.75, 43.06, 59.84) mm, rotated rx 180 ry 0 rz 180 deg; joints [-38.054, -23.942, 90.136, 62.723, 43.909, -54.408]
  MoveL 3334 to (-38.75, 43.06, 59.84) mm, rotated rx 180 ry 0 rz 180 deg; joints [-38.054, -23.942, 90.136, 62.723, 43.909, -54.408]
  Call Extruder(65.20749)
  MoveL 3335 to (-38.57, 42.75, 59.84) mm, rotated rx -180 ry 0 rz -180 deg; joints [-37.977, -23.948, 90.139, 62.656, 43.849, -54.358]
  MoveL 3336 to (-38.57, 42.75, 59.84) mm, rotated rx -180 ry 0 rz -180 deg; joints [-37.977, -23.948, 90.139, 62.656, 43.849, -54.358]
  Call Extruder(65.41482)
  MoveL 3337 to (-38.4, 42.45, 59.84) mm, rotated rx 180 ry 0 rz 180 deg; joints [-37.901, -23.954, 90.143, 62.589, 43.788, -54.308]
  MoveL 3338 to (-38.4, 42.45, 59.84) mm, rotated rx 180 ry 0 rz 180 deg; joints [-37.901, -23.954, 90.143, 62.589, 43.788, -54.308]
  Call Extruder(65.62294)
  MoveL 3339 to (-38.22, 42.15, 59.84) mm, rotated rx 180 ry 0 rz -180 deg; joints [-37.825, -23.96, 90.146, 62.522, 43.727, -54.258]
  MoveL 3340 to (-38.22, 42.15, 59.84) mm, rotated rx 180 ry 0 rz -180 deg; joints [-37.825, -23.96, 90.146, 62.522, 43.727, -54.258]
  Call Extruder(65.74065)
  MoveL 3341 to (-38.12, 41.98, 59.84) mm, rotated rx 180 ry 0 rz 180 deg; joints [-37.782, -23.964, 90.148, 62.485, 43.693, -54.23]
  MoveL 3342 to (-38.12, 41.98, 59.84) mm, rotated rx 180 ry 0 rz 180 deg; joints [-37.782, -23.964, 90.148, 62.485, 43.693, -54.23]
  Call Extruder(66.07350)
  MoveL 3343 to (-37.8, 41.52, 59.84) mm, rotated rx 180 ry 0 rz 180 deg; joints [-37.659, -23.966, 90.149, 62.38, 43.594, -54.153]
  MoveL 3344 to (-37.8, 41.52, 59.84) mm, rotated rx 180 ry 0 rz 180 deg; joints [-37.659, -23.966, 90.149, 62.38, 43.594, -54.153]
  Call Extruder(66.40753)
  MoveL 3345 to (-37.47, 41.07, 59.84) mm, rotated rx 180 ry 0 rz 180 deg; joints [-37.537, -23.968, 90.15, 62.275, 43.495, -54.077]
  MoveL 3346 to (-37.47, 41.07, 59.84) mm, rotated rx 180 ry 0 rz 180 deg; joints [-37.537, -23.968, 90.15, 62.275, 43.495, -54.077]
  Call Extruder(66.57512)
  MoveL 3347 to (-37.3, 40.85, 59.84) mm, rotated rx -180 ry 0 rz -180 deg; joints [-37.475, -23.969, 90.151, 62.222, 43.446, -54.038]
  Call Extruder(67.40443)
  MoveL 3348 to (-36.39, 39.81, 59.84) mm, rotated rx 180 ry 0 rz 180 deg; joints [-37.173, -23.956, 90.144, 61.968, 43.199, -53.857]
  Call Extruder(68.03550)
  MoveL 3349 to (-35.61, 39.11, 59.84) mm, rotated rx 180 ry 0 rz 180 deg; joints [-36.947, -23.93, 90.129, 61.783, 43.01, -53.729]
  MoveL 3350 to (-35.61, 39.11, 59.84) mm, rotated rx 180 ry 0 rz 180 deg; joints [-36.947, -23.93, 90.129, 61.783, 43.01, -53.729]
  Call Extruder(68.23307)
  MoveL 3351 to (-35.35, 38.9, 59.84) mm, rotated rx 180 ry 0 rz 180 deg; joints [-36.876, -23.92, 90.124, 61.726, 42.952, -53.69]
  Call Extruder(68.56709)
  MoveL 3352 to (-34.9, 38.57, 59.84) mm, rotated rx 180 ry 0 rz 180 deg; joints [-36.759, -23.899, 90.112, 61.633, 42.853, -53.627]
  MoveL 3353 to (-34.9, 38.57, 59.84) mm, rotated rx 180 ry 0 rz 180 deg; joints [-36.759, -23.899, 90.112, 61.633, 42.853, -53.627]
  Call Extruder(68.89992)
  MoveL 3354 to (-34.45, 38.24, 59.84) mm, rotated rx 180 ry 0 rz 180 deg; joints [-36.642, -23.877, 90.1, 61.54, 42.754, -53.565]
  MoveL 3355 to (-34.45, 38.24, 59.84) mm, rotated rx 180 ry 0 rz 180 deg; joints [-36.642, -23.877, 90.1, 61.54, 42.754, -53.565]
  Call Extruder(69.07917)
  MoveL 3356 to (-34.21, 38.07, 59.84) mm, rotated rx 180 ry 0 rz 180 deg; joints [-36.579, -23.866, 90.093, 61.49, 42.701, -53.531]
  MoveL 3357 to (-34.21, 38.07, 59.84) mm, rotated rx 180 ry 0 rz 180 deg; joints [-36.579, -23.866, 90.093, 61.49, 42.701, -53.531]
  Call Extruder(69.28728)
  MoveL 3358 to (-33.9, 37.89, 59.84) mm, rotated rx -180 ry 0 rz 180 deg; joints [-36.509, -23.847, 90.083, 61.436, 42.641, -53.496]
  MoveL 3359 to (-33.9, 37.89, 59.84) mm, rotated rx -180 ry 0 rz 180 deg; joints [-36.509, -23.847, 90.083, 61.436, 42.641, -53.496]
  Call Extruder(69.49461)
  MoveL 3360 to (-33.6, 37.71, 59.84) mm, rotated rx -180 ry 0 rz 180 deg; joints [-36.439, -23.829, 90.073, 61.382, 42.58, -53.461]
  MoveL 3361 to (-33.6, 37.71, 59.84) mm, rotated rx -180 ry 0 rz 180 deg; joints [-36.439, -23.829, 90.073, 61.382, 42.58, -53.461]
  Call Extruder(69.70116)
  MoveL 3362 to (-33.29, 37.54, 59.84) mm, rotated rx 180 ry 0 rz 180 deg; joints [-36.368, -23.811, 90.063, 61.327, 42.52, -53.425]
  MoveL 3363 to (-33.29, 37.54, 59.84) mm, rotated rx 180 ry 0 rz 180 deg; joints [-36.368, -23.811, 90.063, 61.327, 42.52, -53.425]
  Call Extruder(69.90693)
  MoveL 3364 to (-32.99, 37.36, 59.84) mm, rotated rx 180 ry 0 rz 180 deg; joints [-36.298, -23.793, 90.053, 61.273, 42.46, -53.39]
  MoveL 3365 to (-32.99, 37.36, 59.84) mm, rotated rx 180 ry 0 rz 180 deg; joints [-36.298, -23.793, 90.053, 61.273, 42.46, -53.39]
  Call Extruder(70.06523)
  MoveL 3366 to (-32.74, 37.26, 59.84) mm, rotated rx -180 ry 0 rz 180 deg; joints [-36.247, -23.775, 90.043, 61.235, 42.415, -53.367]
  MoveL 3367 to (-32.74, 37.26, 59.84) mm, rotated rx -180 ry 0 rz 180 deg; joints [-36.247, -23.775, 90.043, 61.235, 42.415, -53.367]
  Call Extruder(70.22293)
  MoveL 3368 to (-32.49, 37.15, 59.84) mm, rotated rx 180 ry 0 rz 180 deg; joints [-36.196, -23.757, 90.033, 61.198, 42.37, -53.344]
  MoveL 3369 to (-32.49, 37.15, 59.84) mm, rotated rx 180 ry 0 rz 180 deg; joints [-36.196, -23.757, 90.033, 61.198, 42.37, -53.344]
  Call Extruder(70.39301)
  MoveL 3370 to (-32.22, 37.03, 59.84) mm, rotated rx 180 ry 0 rz 180 deg; joints [-36.141, -23.737, 90.022, 61.157, 42.322, -53.319]
  MoveL 3371 to (-32.22, 37.03, 59.84) mm, rotated rx 180 ry 0 rz 180 deg; joints [-36.141, -23.737, 90.022, 61.157, 42.322, -53.319]
  Call Extruder(70.57535)
  MoveL 3372 to (-31.93, 36.91, 59.84) mm, rotated rx 180 ry 0 rz 180 deg; joints [-36.082, -23.716, 90.01, 61.114, 42.27, -53.293]
  MoveL 3373 to (-31.93, 36.91, 59.84) mm, rotated rx 180 ry 0 rz 180 deg; joints [-36.082, -23.716, 90.01, 61.114, 42.27, -53.293]
  Call Extruder(70.75693)
  MoveL 3374 to (-31.64, 36.79, 59.84) mm, rotated rx -180 ry 0 rz 180 deg; joints [-36.023, -23.695, 89.998, 61.071, 42.219, -53.266]
  MoveL 3375 to (-31.64, 36.79, 59.84) mm, rotated rx -180 ry 0 rz 180 deg; joints [-36.023, -23.695, 89.998, 61.071, 42.219, -53.266]
  Call Extruder(70.85628)
  MoveL 3376 to (-31.47, 36.74, 59.84) mm, rotated rx 180 ry 0 rz 180 deg; joints [-35.993, -23.681, 89.99, 61.049, 42.192, -53.254]
  MoveL 3377 to (-31.47, 36.74, 59.84) mm, rotated rx 180 ry 0 rz 180 deg; joints [-35.993, -23.681, 89.99, 61.049, 42.192, -53.254]
  Call Extruder(70.95529)
  MoveL 3378 to (-31.31, 36.69, 59.84) mm, rotated rx 180 ry 0 rz 180 deg; joints [-35.962, -23.668, 89.983, 61.028, 42.164, -53.241]
  MoveL 3379 to (-31.31, 36.69, 59.84) mm, rotated rx 180 ry 0 rz 180 deg; joints [-35.962, -23.668, 89.983, 61.028, 42.164, -53.241]
  Call Extruder(71.05746)
  MoveL 3380 to (-31.14, 36.63, 59.84) mm, rotated rx 180 ry 0 rz -180 deg; joints [-35.931, -23.655, 89.975, 61.005, 42.136, -53.228]
  MoveL 3381 to (-31.14, 36.63, 59.84) mm, rotated rx 180 ry 0 rz -180 deg; joints [-35.931, -23.655, 89.975, 61.005, 42.136, -53.228]
  Call Extruder(71.16269)
  MoveL 3382 to (-30.96, 36.57, 59.84) mm, rotated rx 180 ry 0 rz 180 deg; joints [-35.898, -23.64, 89.967, 60.982, 42.107, -53.215]
  MoveL 3383 to (-30.96, 36.57, 59.84) mm, rotated rx 180 ry 0 rz 180 deg; joints [-35.898, -23.64, 89.967, 60.982, 42.107, -53.215]
  Call Extruder(71.26752)
